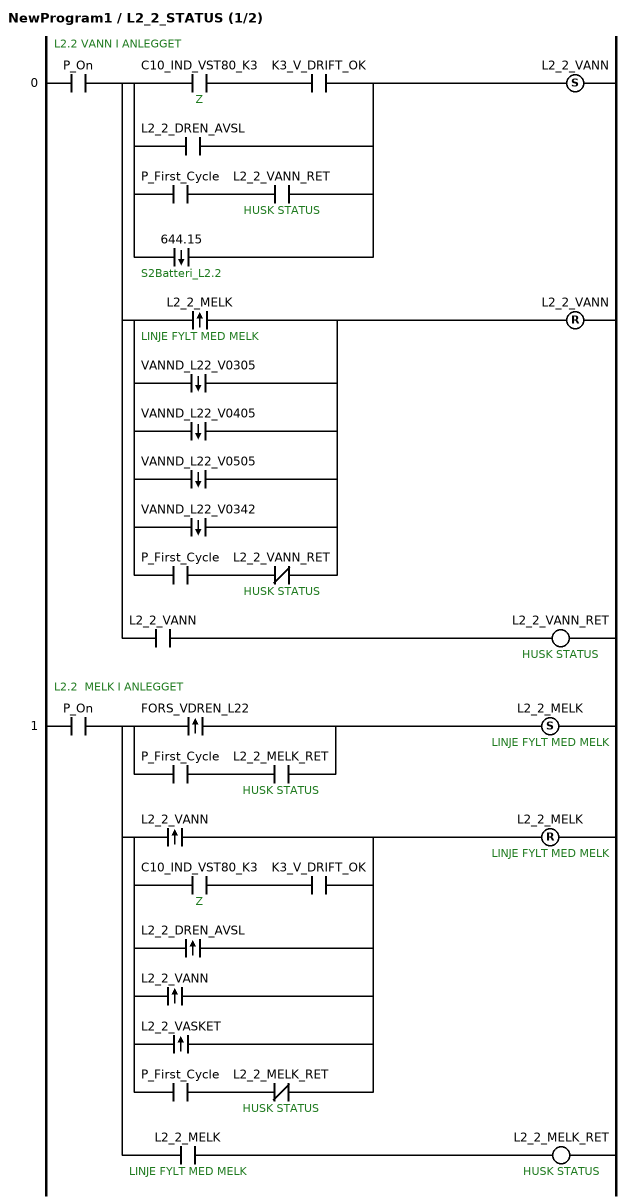
; [picture p816: NewProgram1 / L2_2_STATUS, rungs 0-1]
; rung 0: L2.2 VANN I ANLEGGET
LD P_On
OUT TR0
LD C10_IND_VST80_K3  ; Z
AND K3_V_DRIFT_OK
OR L2_2_DREN_AVSL
LD P_First_Cycle
AND L2_2_VANN_RET  ; HUSK STATUS
ORLD
%OR 644.15  ; S2Batteri_L2.2
ANDLD
SET L2_2_VANN
LD TR0
@LD L2_2_MELK  ; LINJE FYLT MED MELK
%OR VANND_L22_V0305
%OR VANND_L22_V0405
%OR VANND_L22_V0505
%OR VANND_L22_V0342
LD P_First_Cycle
ANDNOT L2_2_VANN_RET  ; HUSK STATUS
ORLD
ANDLD
RSET L2_2_VANN
LD TR0
AND L2_2_VANN
OUT L2_2_VANN_RET  ; HUSK STATUS
; rung 1: L2.2  MELK I ANLEGGET
LD P_On
OUT TR0
@LD FORS_VDREN_L22
LD P_First_Cycle
AND L2_2_MELK_RET  ; HUSK STATUS
ORLD
ANDLD
SET L2_2_MELK  ; LINJE FYLT MED MELK
LD TR0
@LD L2_2_VANN
LD C10_IND_VST80_K3  ; Z
AND K3_V_DRIFT_OK
ORLD
@OR L2_2_DREN_AVSL
@OR L2_2_VANN
@OR L2_2_VASKET
LD P_First_Cycle
ANDNOT L2_2_MELK_RET  ; HUSK STATUS
ORLD
ANDLD
RSET L2_2_MELK  ; LINJE FYLT MED MELK
LD TR0
AND L2_2_MELK  ; LINJE FYLT MED MELK
OUT L2_2_MELK_RET  ; HUSK STATUS

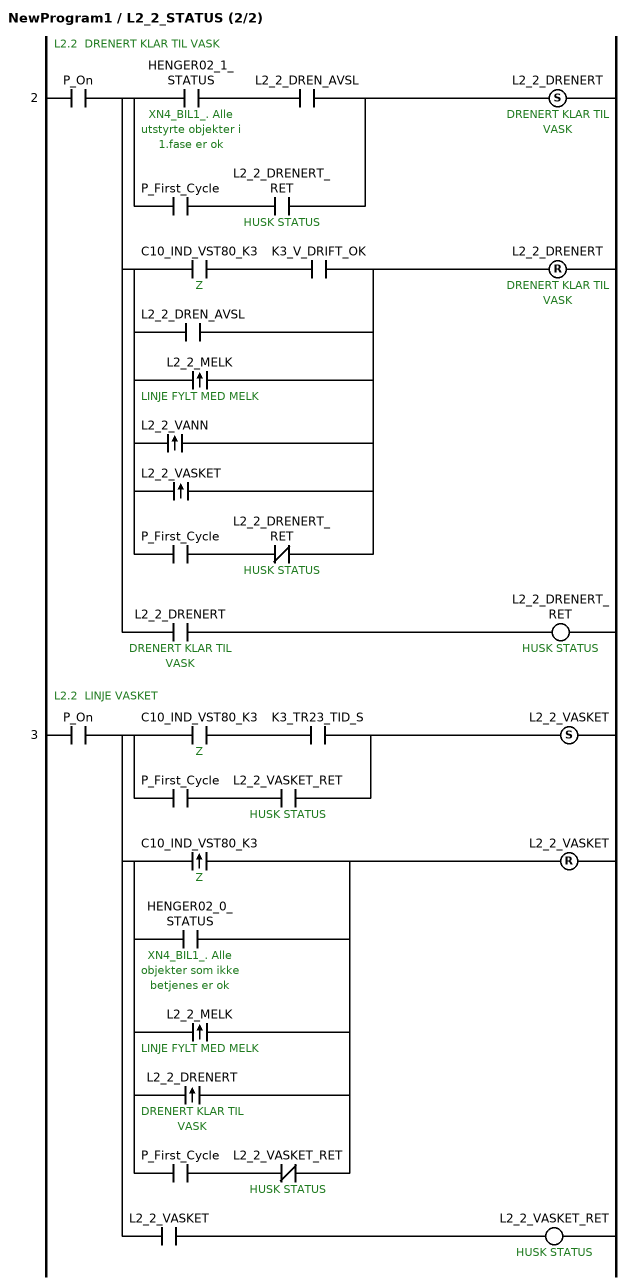
; rung 2: L2.2  DRENERT KLAR TIL VASK
LD P_On
OUT TR0
LD HENGER02_1_STATUS  ; XN4_BIL1_. Alle utstyrte objekter i 1.fase er ok
AND L2_2_DREN_AVSL
LD P_First_Cycle
AND L2_2_DRENERT_RET  ; HUSK STATUS
ORLD
ANDLD
SET L2_2_DRENERT  ; DRENERT KLAR TIL VASK
LD TR0
LD C10_IND_VST80_K3  ; Z
AND K3_V_DRIFT_OK
OR L2_2_DREN_AVSL
@OR L2_2_MELK  ; LINJE FYLT MED MELK
@OR L2_2_VANN
@OR L2_2_VASKET
LD P_First_Cycle
ANDNOT L2_2_DRENERT_RET  ; HUSK STATUS
ORLD
ANDLD
RSET L2_2_DRENERT  ; DRENERT KLAR TIL VASK
LD TR0
AND L2_2_DRENERT  ; DRENERT KLAR TIL VASK
OUT L2_2_DRENERT_RET  ; HUSK STATUS
; rung 3: L2.2  LINJE VASKET
LD P_On
OUT TR0
LD C10_IND_VST80_K3  ; Z
AND K3_TR23_TID_S
LD P_First_Cycle
AND L2_2_VASKET_RET  ; HUSK STATUS
ORLD
ANDLD
SET L2_2_VASKET
LD TR0
@LD C10_IND_VST80_K3  ; Z
OR HENGER02_0_STATUS  ; XN4_BIL1_. Alle objekter som ikke betjenes er ok
@OR L2_2_MELK  ; LINJE FYLT MED MELK
@OR L2_2_DRENERT  ; DRENERT KLAR TIL VASK
LD P_First_Cycle
ANDNOT L2_2_VASKET_RET  ; HUSK STATUS
ORLD
ANDLD
RSET L2_2_VASKET
LD TR0
AND L2_2_VASKET
OUT L2_2_VASKET_RET  ; HUSK STATUS

### Section L2_2_FUNKSJONER

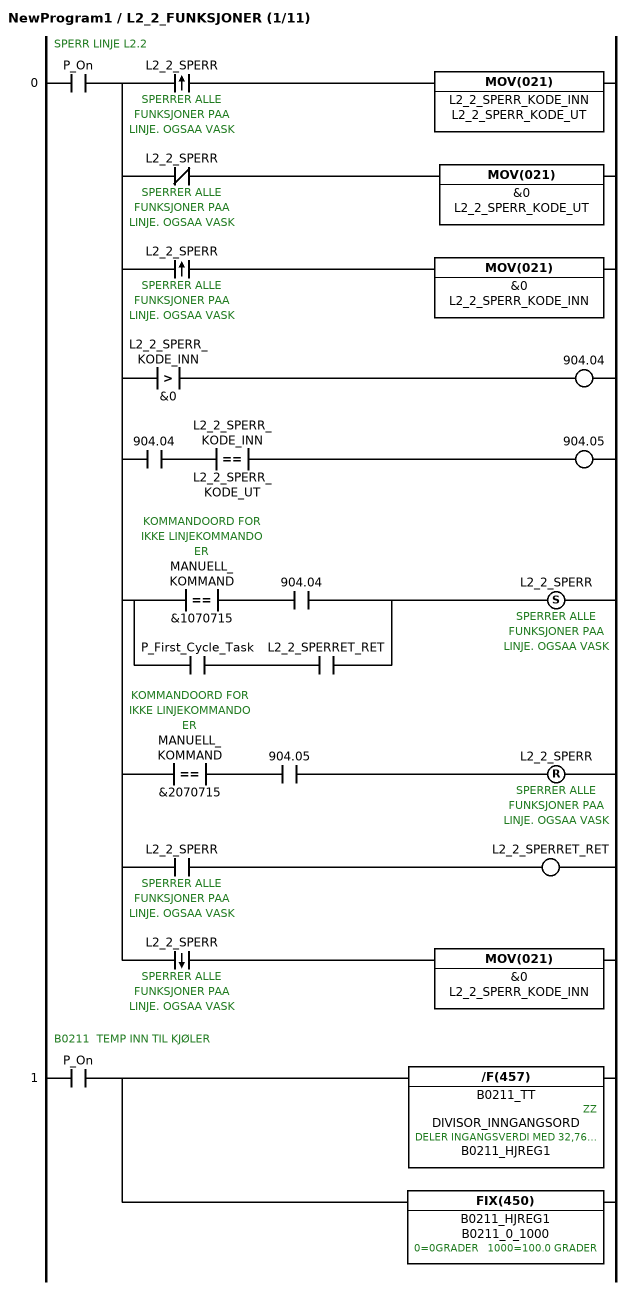
; rung 0: SPERR LINJE L2.2
LD P_On
OUT TR0
@AND L2_2_SPERR  ; SPERRER ALLE FUNKSJONER PAA LINJE. OGSAA VASK
MOV(021) L2_2_SPERR_KODE_INN L2_2_SPERR_KODE_UT
LD TR0
ANDNOT L2_2_SPERR  ; SPERRER ALLE FUNKSJONER PAA LINJE. OGSAA VASK
MOV(021) &0 L2_2_SPERR_KODE_UT
LD TR0
@AND L2_2_SPERR  ; SPERRER ALLE FUNKSJONER PAA LINJE. OGSAA VASK
MOV(021) &0 L2_2_SPERR_KODE_INN
LD TR0
AND>(320) L2_2_SPERR_KODE_INN &0
OUT 904.04
LD TR0
AND 904.04
AND=(300) L2_2_SPERR_KODE_INN L2_2_SPERR_KODE_UT
OUT 904.05
LD TR0
LD=L(301) MANUELL_KOMMAND &1070715  ; KOMMANDOORD FOR IKKE LINJEKOMMANDOER
AND 904.04
LD P_First_Cycle_Task
AND L2_2_SPERRET_RET
ORLD
ANDLD
SET L2_2_SPERR  ; SPERRER ALLE FUNKSJONER PAA LINJE. OGSAA VASK
LD TR0
AND=L(301) MANUELL_KOMMAND &2070715  ; KOMMANDOORD FOR IKKE LINJEKOMMANDOER
AND 904.05
RSET L2_2_SPERR  ; SPERRER ALLE FUNKSJONER PAA LINJE. OGSAA VASK
LD TR0
AND L2_2_SPERR  ; SPERRER ALLE FUNKSJONER PAA LINJE. OGSAA VASK
OUT L2_2_SPERRET_RET
LD TR0
%AND L2_2_SPERR  ; SPERRER ALLE FUNKSJONER PAA LINJE. OGSAA VASK
MOV(021) &0 L2_2_SPERR_KODE_INN
; rung 1: B0211  TEMP INN TIL KJØLER
LD P_On
/F(457) B0211_TT DIVISOR_INNGANGSORD B0211_HJREG1  ; ZZ, DELER INGANGSVERDI MED 32,760 FOR OMREGNING TIL 0-1000
FIX(450) B0211_HJREG1 B0211_0_1000  ; 0=0GRADER   1000=100.0 GRADER

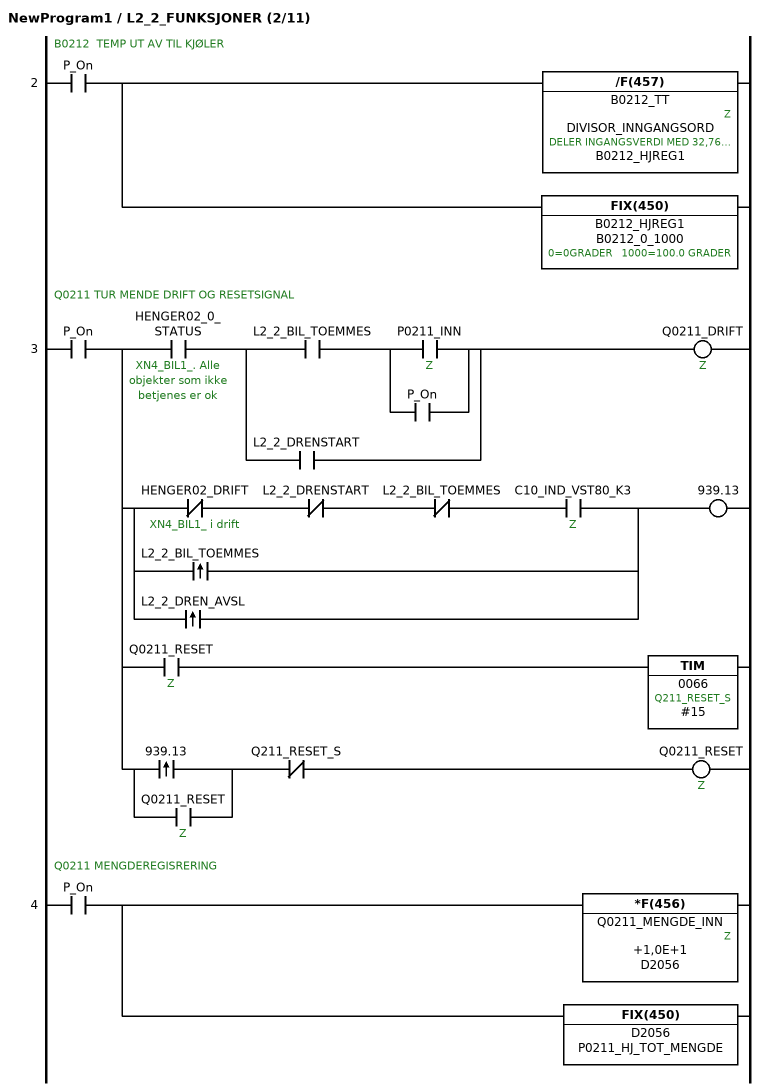
; rung 2: B0212  TEMP UT AV TIL KJØLER
LD P_On
/F(457) B0212_TT DIVISOR_INNGANGSORD B0212_HJREG1  ; Z, DELER INGANGSVERDI MED 32,760 FOR OMREGNING TIL 0-1000
FIX(450) B0212_HJREG1 B0212_0_1000  ; 0=0GRADER   1000=100.0 GRADER
; rung 3: Q0211 TUR MENDE DRIFT OG RESETSIGNAL
LD P_On
OUT TR0
AND HENGER02_0_STATUS  ; XN4_BIL1_. Alle objekter som ikke betjenes er ok
LD L2_2_BIL_TOEMMES
LD P0211_INN  ; Z
OR P_On
ANDLD
OR L2_2_DRENSTART
ANDLD
OUT Q0211_DRIFT  ; Z
LD TR0
LDNOT HENGER02_DRIFT  ; XN4_BIL1_ i drift
ANDNOT L2_2_DRENSTART
ANDNOT L2_2_BIL_TOEMMES
AND C10_IND_VST80_K3  ; Z
@OR L2_2_BIL_TOEMMES
@OR L2_2_DREN_AVSL
ANDLD
OUT 939.13
LD TR0
AND Q0211_RESET  ; Z
TIM 0066 #15  ; Q211_RESET_S
LD TR0
@LD 939.13
OR Q0211_RESET  ; Z
ANDLD
ANDNOT Q211_RESET_S
OUT Q0211_RESET  ; Z
; rung 4: Q0211 MENGDEREGISRERING
LD P_On
*F(456) Q0211_MENGDE_INN +1,0E+1 D2056  ; Z
FIX(450) D2056 P0211_HJ_TOT_MENGDE

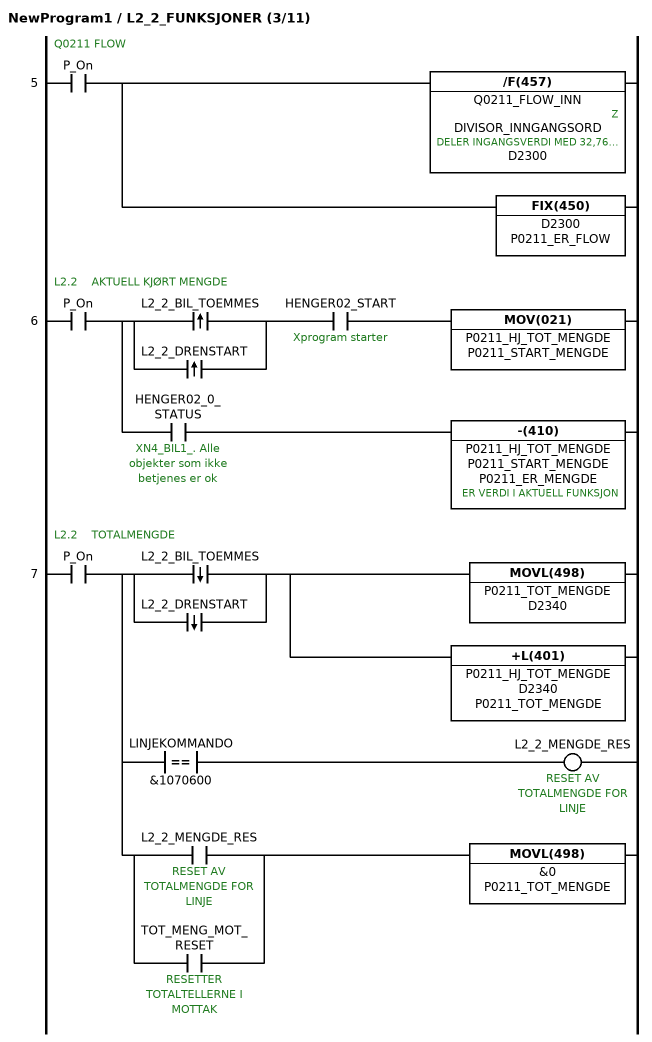
; rung 5: Q0211 FLOW
LD P_On
/F(457) Q0211_FLOW_INN DIVISOR_INNGANGSORD D2300  ; Z, DELER INGANGSVERDI MED 32,760 FOR OMREGNING TIL 0-1000
FIX(450) D2300 P0211_ER_FLOW
; rung 6: L2.2    AKTUELL KJØRT MENGDE
LD P_On
OUT TR0
@LD L2_2_BIL_TOEMMES
@OR L2_2_DRENSTART
ANDLD
AND HENGER02_START  ; Xprogram starter
MOV(021) P0211_HJ_TOT_MENGDE P0211_START_MENGDE
LD TR0
AND HENGER02_0_STATUS  ; XN4_BIL1_. Alle objekter som ikke betjenes er ok
-(410) P0211_HJ_TOT_MENGDE P0211_START_MENGDE P0211_ER_MENGDE  ; ER VERDI I AKTUELL FUNKSJON
; rung 7: L2.2    TOTALMENGDE
LD P_On
OUT TR0
%LD L2_2_BIL_TOEMMES
%OR L2_2_DRENSTART
ANDLD
MOVL(498) P0211_TOT_MENGDE D2340
+L(401) P0211_HJ_TOT_MENGDE D2340 P0211_TOT_MENGDE
LD TR0
AND=L(301) LINJEKOMMANDO &1070600
OUT L2_2_MENGDE_RES  ; RESET AV  TOTALMENGDE FOR LINJE
LD TR0
LD L2_2_MENGDE_RES  ; RESET AV  TOTALMENGDE FOR LINJE
OR TOT_MENG_MOT_RESET  ; RESETTER TOTALTELLERNE I MOTTAK
ANDLD
MOVL(498) &0 P0211_TOT_MENGDE

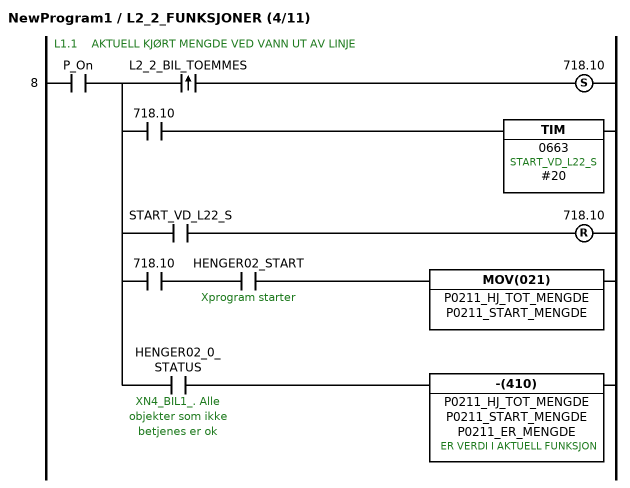
; rung 8: L1.1    AKTUELL KJØRT MENGDE VED VANN UT AV LINJE
LD P_On
OUT TR0
@AND L2_2_BIL_TOEMMES
SET 718.10
LD TR0
AND 718.10
TIM 0663 #20  ; START_VD_L22_S
LD TR0
AND START_VD_L22_S
RSET 718.10
LD TR0
AND 718.10
AND HENGER02_START  ; Xprogram starter
MOV(021) P0211_HJ_TOT_MENGDE P0211_START_MENGDE
LD TR0
AND HENGER02_0_STATUS  ; XN4_BIL1_. Alle objekter som ikke betjenes er ok
-(410) P0211_HJ_TOT_MENGDE P0211_START_MENGDE P0211_ER_MENGDE  ; ER VERDI I AKTUELL FUNKSJON

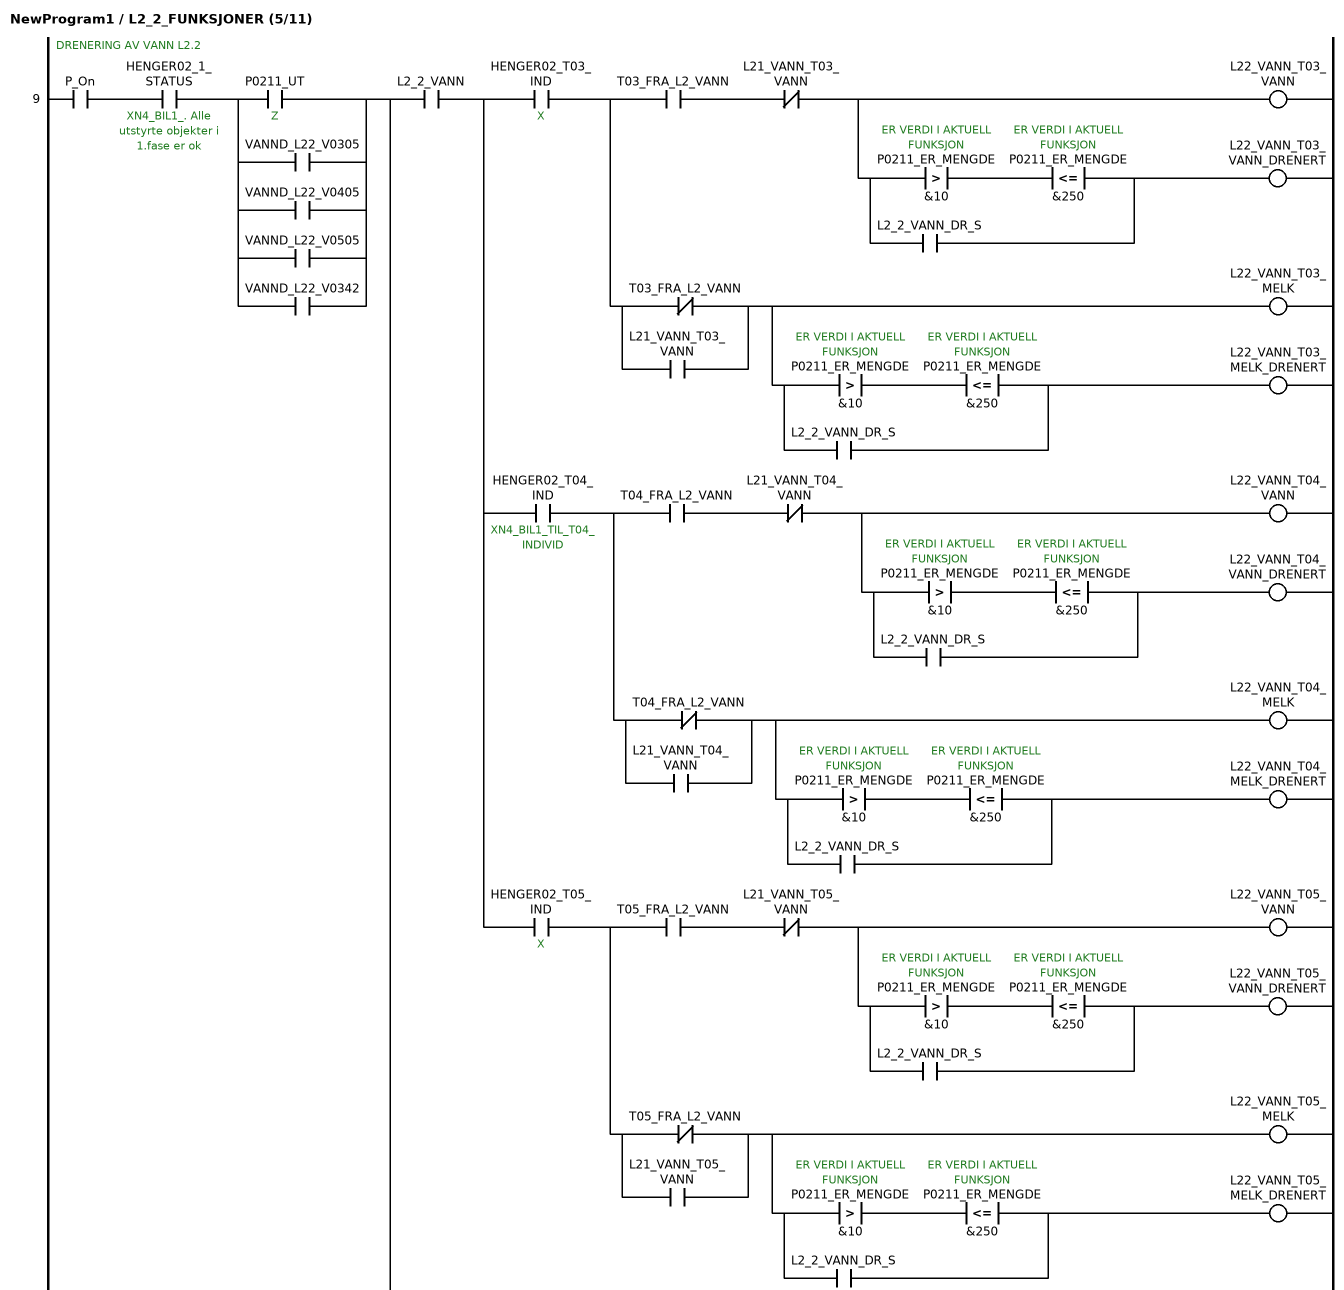

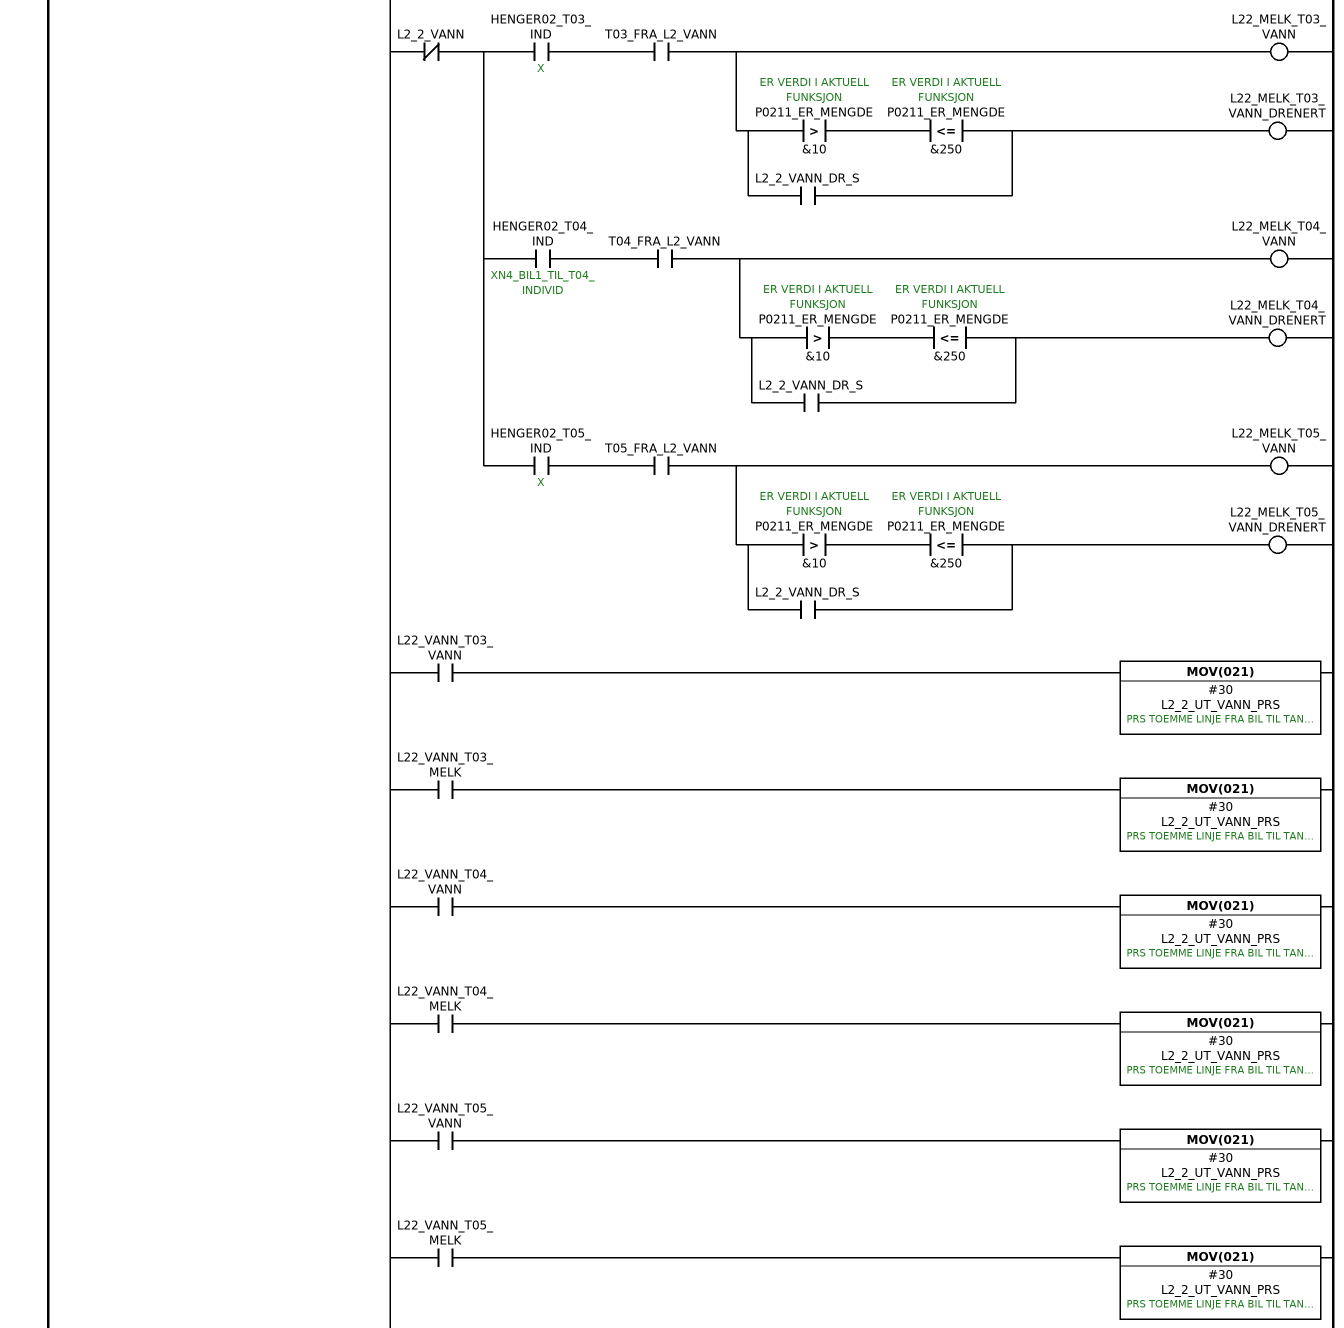

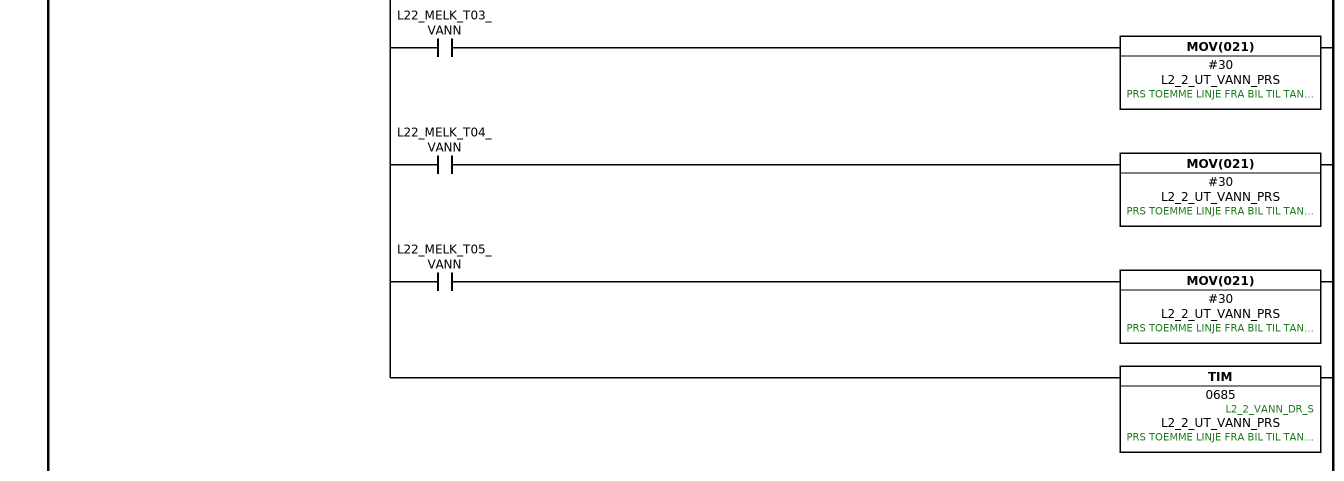
; rung 9: DRENERING AV VANN L2.2
LD P_On
AND HENGER02_1_STATUS  ; XN4_BIL1_. Alle utstyrte objekter i 1.fase er ok
LD P0211_UT  ; Z
OR VANND_L22_V0305
OR VANND_L22_V0405
OR VANND_L22_V0505
OR VANND_L22_V0342
ANDLD
OUT TR0
AND L2_2_VANN
OUT TR1
AND HENGER02_T03_IND  ; X
OUT TR2
AND T03_FRA_L2_VANN
ANDNOT L21_VANN_T03_VANN
OUT L22_VANN_T03_VANN
LD>(320) P0211_ER_MENGDE &10  ; ER VERDI I AKTUELL FUNKSJON
AND<=(315) P0211_ER_MENGDE &250  ; ER VERDI I AKTUELL FUNKSJON
OR L2_2_VANN_DR_S
ANDLD
OUT L22_VANN_T03_VANN_DRENERT
LD TR2
LDNOT T03_FRA_L2_VANN
OR L21_VANN_T03_VANN
ANDLD
OUT L22_VANN_T03_MELK
LD>(320) P0211_ER_MENGDE &10  ; ER VERDI I AKTUELL FUNKSJON
AND<=(315) P0211_ER_MENGDE &250  ; ER VERDI I AKTUELL FUNKSJON
OR L2_2_VANN_DR_S
ANDLD
OUT L22_VANN_T03_MELK_DRENERT
LD TR1
AND HENGER02_T04_IND  ; XN4_BIL1_TIL_T04_INDIVID
OUT TR2
AND T04_FRA_L2_VANN
ANDNOT L21_VANN_T04_VANN
OUT L22_VANN_T04_VANN
LD>(320) P0211_ER_MENGDE &10  ; ER VERDI I AKTUELL FUNKSJON
AND<=(315) P0211_ER_MENGDE &250  ; ER VERDI I AKTUELL FUNKSJON
OR L2_2_VANN_DR_S
ANDLD
OUT L22_VANN_T04_VANN_DRENERT
LD TR2
LDNOT T04_FRA_L2_VANN
OR L21_VANN_T04_VANN
ANDLD
OUT L22_VANN_T04_MELK
LD>(320) P0211_ER_MENGDE &10  ; ER VERDI I AKTUELL FUNKSJON
AND<=(315) P0211_ER_MENGDE &250  ; ER VERDI I AKTUELL FUNKSJON
OR L2_2_VANN_DR_S
ANDLD
OUT L22_VANN_T04_MELK_DRENERT
LD TR1
AND HENGER02_T05_IND  ; X
OUT TR1
AND T05_FRA_L2_VANN
ANDNOT L21_VANN_T05_VANN
OUT L22_VANN_T05_VANN
LD>(320) P0211_ER_MENGDE &10  ; ER VERDI I AKTUELL FUNKSJON
AND<=(315) P0211_ER_MENGDE &250  ; ER VERDI I AKTUELL FUNKSJON
OR L2_2_VANN_DR_S
ANDLD
OUT L22_VANN_T05_VANN_DRENERT
LD TR1
LDNOT T05_FRA_L2_VANN
OR L21_VANN_T05_VANN
ANDLD
OUT L22_VANN_T05_MELK
LD>(320) P0211_ER_MENGDE &10  ; ER VERDI I AKTUELL FUNKSJON
AND<=(315) P0211_ER_MENGDE &250  ; ER VERDI I AKTUELL FUNKSJON
OR L2_2_VANN_DR_S
ANDLD
OUT L22_VANN_T05_MELK_DRENERT
LD TR0
ANDNOT L2_2_VANN
OUT TR1
AND HENGER02_T03_IND  ; X
AND T03_FRA_L2_VANN
OUT L22_MELK_T03_VANN
LD>(320) P0211_ER_MENGDE &10  ; ER VERDI I AKTUELL FUNKSJON
AND<=(315) P0211_ER_MENGDE &250  ; ER VERDI I AKTUELL FUNKSJON
OR L2_2_VANN_DR_S
ANDLD
OUT L22_MELK_T03_VANN_DRENERT
LD TR1
AND HENGER02_T04_IND  ; XN4_BIL1_TIL_T04_INDIVID
AND T04_FRA_L2_VANN
OUT L22_MELK_T04_VANN
LD>(320) P0211_ER_MENGDE &10  ; ER VERDI I AKTUELL FUNKSJON
AND<=(315) P0211_ER_MENGDE &250  ; ER VERDI I AKTUELL FUNKSJON
OR L2_2_VANN_DR_S
ANDLD
OUT L22_MELK_T04_VANN_DRENERT
LD TR1
AND HENGER02_T05_IND  ; X
AND T05_FRA_L2_VANN
OUT L22_MELK_T05_VANN
LD>(320) P0211_ER_MENGDE &10  ; ER VERDI I AKTUELL FUNKSJON
AND<=(315) P0211_ER_MENGDE &250  ; ER VERDI I AKTUELL FUNKSJON
OR L2_2_VANN_DR_S
ANDLD
OUT L22_MELK_T05_VANN_DRENERT
LD TR0
AND L22_VANN_T03_VANN
MOV(021) #30 L2_2_UT_VANN_PRS  ; PRS TOEMME LINJE FRA BIL TIL TANK FOR VANN
LD TR0
AND L22_VANN_T03_MELK
MOV(021) #30 L2_2_UT_VANN_PRS  ; PRS TOEMME LINJE FRA BIL TIL TANK FOR VANN
LD TR0
AND L22_VANN_T04_VANN
MOV(021) #30 L2_2_UT_VANN_PRS  ; PRS TOEMME LINJE FRA BIL TIL TANK FOR VANN
LD TR0
AND L22_VANN_T04_MELK
MOV(021) #30 L2_2_UT_VANN_PRS  ; PRS TOEMME LINJE FRA BIL TIL TANK FOR VANN
LD TR0
AND L22_VANN_T05_VANN
MOV(021) #30 L2_2_UT_VANN_PRS  ; PRS TOEMME LINJE FRA BIL TIL TANK FOR VANN
LD TR0
AND L22_VANN_T05_MELK
MOV(021) #30 L2_2_UT_VANN_PRS  ; PRS TOEMME LINJE FRA BIL TIL TANK FOR VANN
LD TR0
AND L22_MELK_T03_VANN
MOV(021) #30 L2_2_UT_VANN_PRS  ; PRS TOEMME LINJE FRA BIL TIL TANK FOR VANN
LD TR0
AND L22_MELK_T04_VANN
MOV(021) #30 L2_2_UT_VANN_PRS  ; PRS TOEMME LINJE FRA BIL TIL TANK FOR VANN
LD TR0
AND L22_MELK_T05_VANN
MOV(021) #30 L2_2_UT_VANN_PRS  ; PRS TOEMME LINJE FRA BIL TIL TANK FOR VANN
LD TR0
TIM 0685 L2_2_UT_VANN_PRS  ; PRS TOEMME LINJE FRA BIL TIL TANK FOR VANN, L2_2_VANN_DR_S

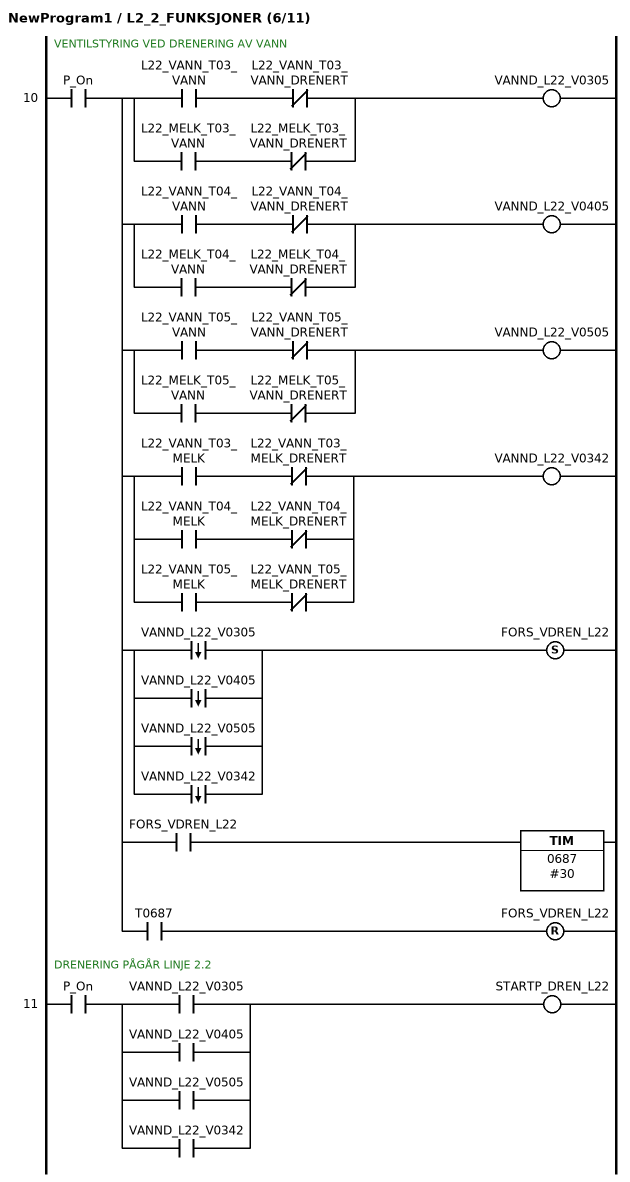
; rung 10: VENTILSTYRING VED DRENERING AV VANN
LD P_On
OUT TR0
LD L22_VANN_T03_VANN
ANDNOT L22_VANN_T03_VANN_DRENERT
LD L22_MELK_T03_VANN
ANDNOT L22_MELK_T03_VANN_DRENERT
ORLD
ANDLD
OUT VANND_L22_V0305
LD TR0
LD L22_VANN_T04_VANN
ANDNOT L22_VANN_T04_VANN_DRENERT
LD L22_MELK_T04_VANN
ANDNOT L22_MELK_T04_VANN_DRENERT
ORLD
ANDLD
OUT VANND_L22_V0405
LD TR0
LD L22_VANN_T05_VANN
ANDNOT L22_VANN_T05_VANN_DRENERT
LD L22_MELK_T05_VANN
ANDNOT L22_MELK_T05_VANN_DRENERT
ORLD
ANDLD
OUT VANND_L22_V0505
LD TR0
LD L22_VANN_T03_MELK
ANDNOT L22_VANN_T03_MELK_DRENERT
LD L22_VANN_T04_MELK
ANDNOT L22_VANN_T04_MELK_DRENERT
ORLD
LD L22_VANN_T05_MELK
ANDNOT L22_VANN_T05_MELK_DRENERT
ORLD
ANDLD
OUT VANND_L22_V0342
LD TR0
%LD VANND_L22_V0305
%OR VANND_L22_V0405
%OR VANND_L22_V0505
%OR VANND_L22_V0342
ANDLD
SET FORS_VDREN_L22
LD TR0
AND FORS_VDREN_L22
TIM 0687 #30
LD TR0
AND T0687
RSET FORS_VDREN_L22
; rung 11: DRENERING PÅGÅR LINJE 2.2
LD P_On
LD VANND_L22_V0305
OR VANND_L22_V0405
OR VANND_L22_V0505
OR VANND_L22_V0342
ANDLD
OUT STARTP_DREN_L22

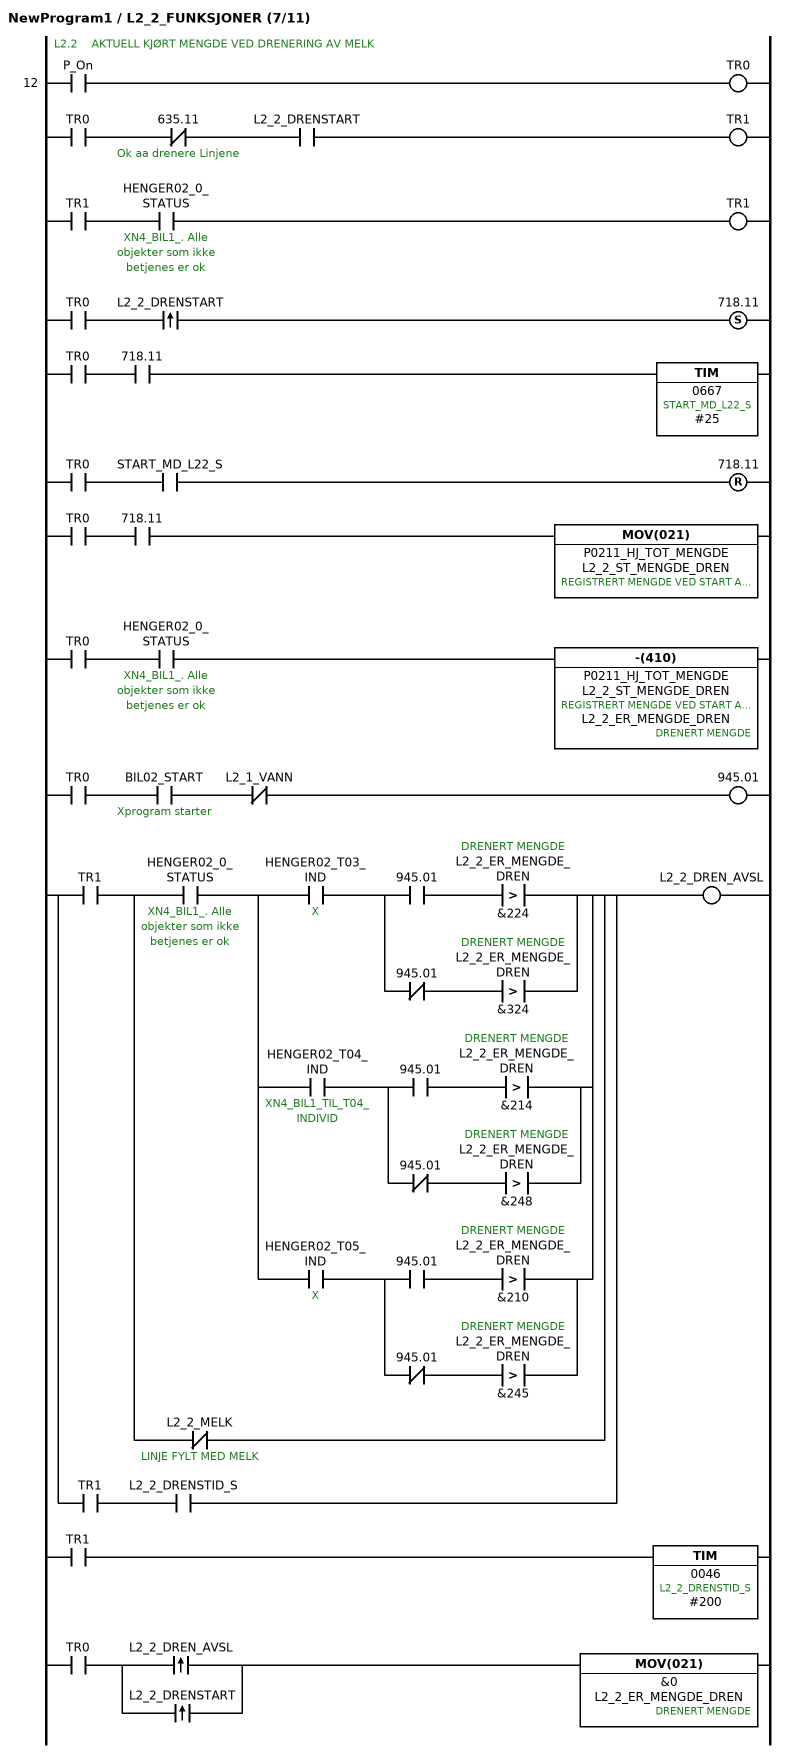
; rung 12: L2.2    AKTUELL KJØRT MENGDE VED DRENERING AV MELK
LD P_On
OUT TR0
@AND L2_2_DRENSTART
SET 718.11
LD TR0
AND 718.11
TIM 0667 #25  ; START_MD_L22_S
LD TR0
AND START_MD_L22_S
RSET 718.11
LD TR0
AND 718.11
MOV(021) P0211_HJ_TOT_MENGDE L2_2_ST_MENGDE_DREN  ; REGISTRERT MENGDE VED START AV DREN.
LD TR0
AND HENGER02_0_STATUS  ; XN4_BIL1_. Alle objekter som ikke betjenes er ok
-(410) P0211_HJ_TOT_MENGDE L2_2_ST_MENGDE_DREN L2_2_ER_MENGDE_DREN  ; REGISTRERT MENGDE VED START AV DREN., DRENERT MENGDE
LD TR0
AND BIL02_START  ; Xprogram starter
ANDNOT L2_1_VANN
OUT 945.01
LD TR0
ANDNOT 635.11  ; Ok aa drenere Linjene
AND L2_2_DRENSTART
OUT TR1
LD HENGER02_0_STATUS  ; XN4_BIL1_. Alle objekter som ikke betjenes er ok
LD HENGER02_T03_IND  ; X
LD 945.01
AND>(320) L2_2_ER_MENGDE_DREN &224  ; DRENERT MENGDE
LDNOT 945.01
AND>(320) L2_2_ER_MENGDE_DREN &324  ; DRENERT MENGDE
ORLD
ANDLD
LD HENGER02_T04_IND  ; XN4_BIL1_TIL_T04_INDIVID
LD 945.01
AND>(320) L2_2_ER_MENGDE_DREN &214  ; DRENERT MENGDE
LDNOT 945.01
AND>(320) L2_2_ER_MENGDE_DREN &248  ; DRENERT MENGDE
ORLD
ANDLD
ORLD
LD HENGER02_T05_IND  ; X
LD 945.01
AND>(320) L2_2_ER_MENGDE_DREN &210  ; DRENERT MENGDE
LDNOT 945.01
AND>(320) L2_2_ER_MENGDE_DREN &245  ; DRENERT MENGDE
ORLD
ANDLD
ORLD
ANDLD
ORNOT L2_2_MELK  ; LINJE FYLT MED MELK
ANDLD
LD TR1
AND HENGER02_0_STATUS  ; XN4_BIL1_. Alle objekter som ikke betjenes er ok
OUT TR1
AND L2_2_DRENSTID_S
ORLD
OUT L2_2_DREN_AVSL
LD TR1
TIM 0046 #200  ; L2_2_DRENSTID_S
LD TR0
@LD L2_2_DREN_AVSL
@OR L2_2_DRENSTART
ANDLD
MOV(021) &0 L2_2_ER_MENGDE_DREN  ; DRENERT MENGDE

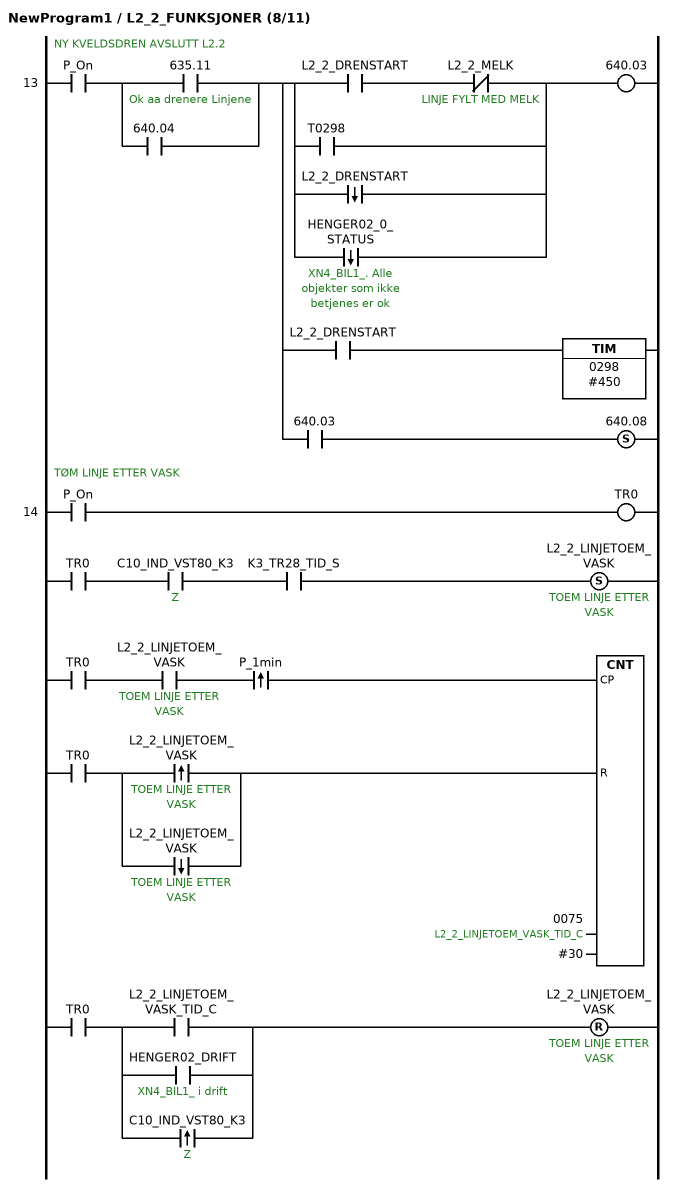
; rung 13: NY KVELDSDREN AVSLUTT L2.2
LD P_On
LD 635.11  ; Ok aa drenere Linjene
OR 640.04
ANDLD
OUT TR0
LD L2_2_DRENSTART
ANDNOT L2_2_MELK  ; LINJE FYLT MED MELK
OR T0298
%OR L2_2_DRENSTART
%OR HENGER02_0_STATUS  ; XN4_BIL1_. Alle objekter som ikke betjenes er ok
ANDLD
OUT 640.03
LD TR0
AND L2_2_DRENSTART
TIM 0298 #450
LD TR0
AND 640.03
SET 640.08
; rung 14: TØM LINJE ETTER VASK
LD P_On
OUT TR0
AND C10_IND_VST80_K3  ; Z
AND K3_TR28_TID_S
SET L2_2_LINJETOEM_VASK  ; TOEM LINJE ETTER VASK
LD TR0
AND L2_2_LINJETOEM_VASK  ; TOEM LINJE ETTER VASK
@AND P_1min
LD TR0
@LD L2_2_LINJETOEM_VASK  ; TOEM LINJE ETTER VASK
%OR L2_2_LINJETOEM_VASK  ; TOEM LINJE ETTER VASK
ANDLD
CNT 0075 #30  ; L2_2_LINJETOEM_VASK_TID_C
LD TR0
LD L2_2_LINJETOEM_VASK_TID_C
OR HENGER02_DRIFT  ; XN4_BIL1_ i drift
@OR C10_IND_VST80_K3  ; Z
ANDLD
RSET L2_2_LINJETOEM_VASK  ; TOEM LINJE ETTER VASK

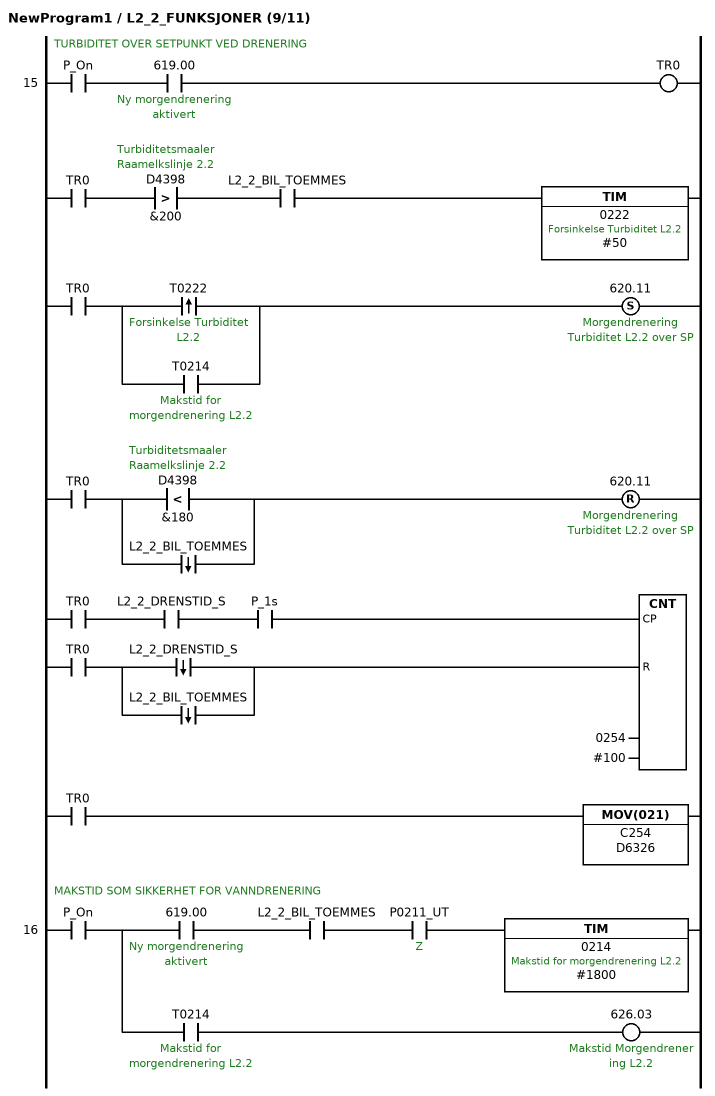
; rung 15: TURBIDITET OVER SETPUNKT VED DRENERING
LD P_On
AND 619.00  ; Ny morgendrenering aktivert
OUT TR0
AND>(320) D4398 &200  ; Turbiditetsmaaler Raamelkslinje 2.2
AND L2_2_BIL_TOEMMES
TIM 0222 #50  ; Forsinkelse Turbiditet L2.2
LD TR0
@LD T0222  ; Forsinkelse Turbiditet L2.2
OR T0214  ; Makstid for morgendrenering L2.2
ANDLD
SET 620.11  ; Morgendrenering Turbiditet L2.2 over SP
LD TR0
LD<(310) D4398 &180  ; Turbiditetsmaaler Raamelkslinje 2.2
%OR L2_2_BIL_TOEMMES
ANDLD
RSET 620.11  ; Morgendrenering Turbiditet L2.2 over SP
LD TR0
AND L2_2_DRENSTID_S
AND P_1s
LD TR0
%LD L2_2_DRENSTID_S
%OR L2_2_BIL_TOEMMES
ANDLD
CNT 0254 #100
LD TR0
MOV(021) C254 D6326
; rung 16: MAKSTID SOM SIKKERHET FOR VANNDRENERING
LD P_On
OUT TR0
AND 619.00  ; Ny morgendrenering aktivert
AND L2_2_BIL_TOEMMES
AND P0211_UT  ; Z
TIM 0214 #1800  ; Makstid for morgendrenering L2.2
LD TR0
AND T0214  ; Makstid for morgendrenering L2.2
OUT 626.03  ; Makstid Morgendrenering L2.2

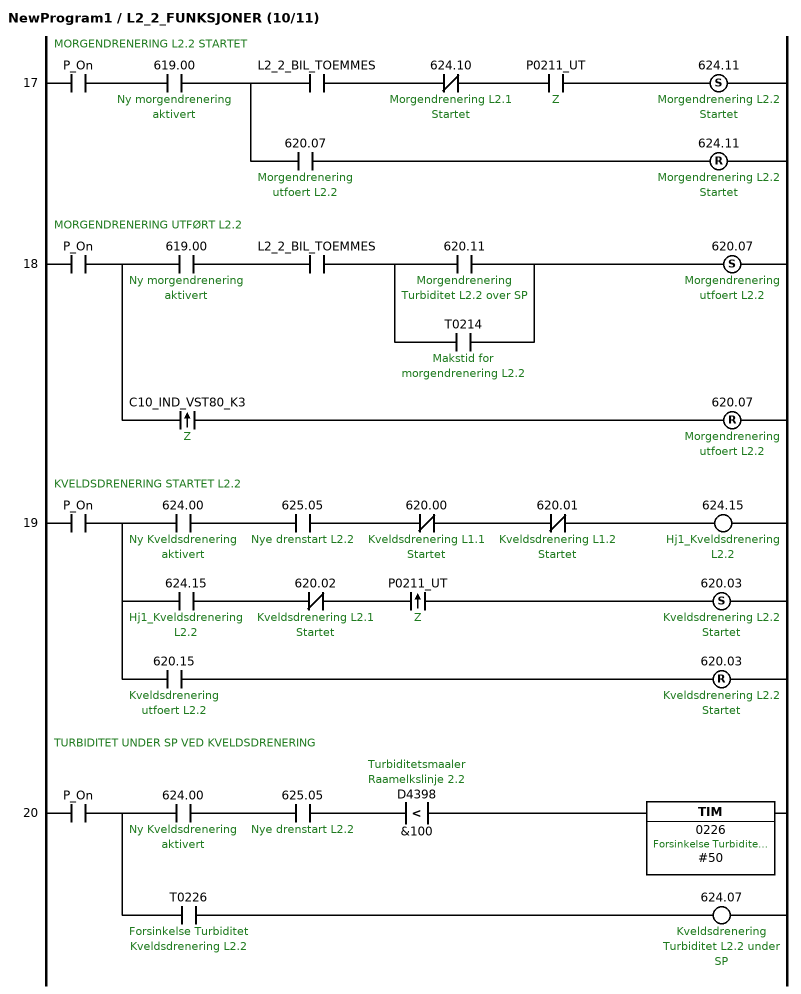
; rung 17: MORGENDRENERING L2.2 STARTET
LD P_On
AND 619.00  ; Ny morgendrenering aktivert
OUT TR0
AND L2_2_BIL_TOEMMES
ANDNOT 624.10  ; Morgendrenering L2.1 Startet
AND P0211_UT  ; Z
SET 624.11  ; Morgendrenering L2.2 Startet
LD TR0
AND 620.07  ; Morgendrenering utfoert L2.2
RSET 624.11  ; Morgendrenering L2.2 Startet
; rung 18: MORGENDRENERING UTFØRT L2.2
LD P_On
OUT TR0
AND 619.00  ; Ny morgendrenering aktivert
AND L2_2_BIL_TOEMMES
LD 620.11  ; Morgendrenering Turbiditet L2.2 over SP
OR T0214  ; Makstid for morgendrenering L2.2
ANDLD
SET 620.07  ; Morgendrenering utfoert L2.2
LD TR0
@AND C10_IND_VST80_K3  ; Z
RSET 620.07  ; Morgendrenering utfoert L2.2
; rung 19: KVELDSDRENERING STARTET L2.2
LD P_On
OUT TR0
AND 624.00  ; Ny Kveldsdrenering aktivert
AND 625.05  ; Nye drenstart L2.2
ANDNOT 620.00  ; Kveldsdrenering L1.1 Startet
ANDNOT 620.01  ; Kveldsdrenering L1.2 Startet
OUT 624.15  ; Hj1_Kveldsdrenering L2.2
LD TR0
AND 624.15  ; Hj1_Kveldsdrenering L2.2
ANDNOT 620.02  ; Kveldsdrenering L2.1 Startet
@AND P0211_UT  ; Z
SET 620.03  ; Kveldsdrenering L2.2 Startet
LD TR0
AND 620.15  ; Kveldsdrenering utfoert L2.2
RSET 620.03  ; Kveldsdrenering L2.2 Startet
; rung 20: TURBIDITET UNDER SP VED KVELDSDRENERING
LD P_On
OUT TR0
AND 624.00  ; Ny Kveldsdrenering aktivert
AND 625.05  ; Nye drenstart L2.2
AND<(310) D4398 &100  ; Turbiditetsmaaler Raamelkslinje 2.2
TIM 0226 #50  ; Forsinkelse Turbiditet Kveldsdrenering L2.2
LD TR0
AND T0226  ; Forsinkelse Turbiditet Kveldsdrenering L2.2
OUT 624.07  ; Kveldsdrenering Turbiditet L2.2 under SP

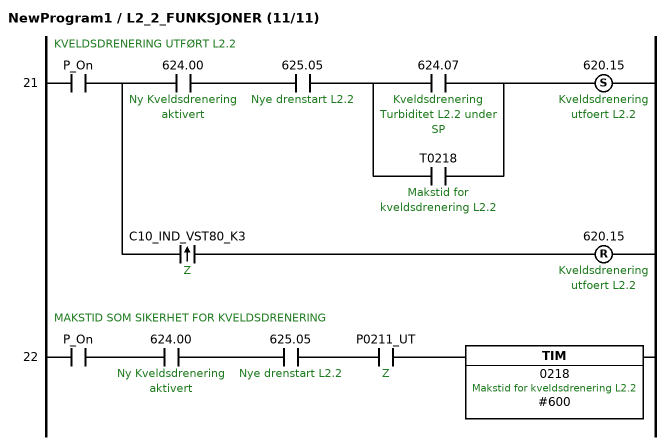
; rung 21: KVELDSDRENERING UTFØRT L2.2
LD P_On
OUT TR0
AND 624.00  ; Ny Kveldsdrenering aktivert
AND 625.05  ; Nye drenstart L2.2
LD 624.07  ; Kveldsdrenering Turbiditet L2.2 under SP
OR T0218  ; Makstid for kveldsdrenering L2.2
ANDLD
SET 620.15  ; Kveldsdrenering utfoert L2.2
LD TR0
@AND C10_IND_VST80_K3  ; Z
RSET 620.15  ; Kveldsdrenering utfoert L2.2
; rung 22: MAKSTID SOM SIKERHET FOR KVELDSDRENERING
LD P_On
AND 624.00  ; Ny Kveldsdrenering aktivert
AND 625.05  ; Nye drenstart L2.2
AND P0211_UT  ; Z
TIM 0218 #600  ; Makstid for kveldsdrenering L2.2

### Section L1_1_TIL_L2_2_FELLESFUNKSJONER

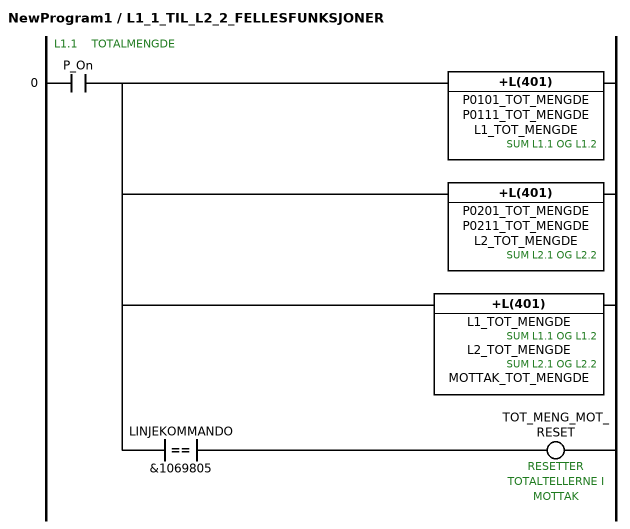
; rung 0: L1.1    TOTALMENGDE
LD P_On
+L(401) P0101_TOT_MENGDE P0111_TOT_MENGDE L1_TOT_MENGDE  ; SUM L1.1 OG L1.2
+L(401) P0201_TOT_MENGDE P0211_TOT_MENGDE L2_TOT_MENGDE  ; SUM L2.1 OG L2.2
+L(401) L1_TOT_MENGDE L2_TOT_MENGDE MOTTAK_TOT_MENGDE  ; SUM L1.1 OG L1.2, SUM L2.1 OG L2.2
AND=L(301) LINJEKOMMANDO &1069805
OUT TOT_MENG_MOT_RESET  ; RESETTER TOTALTELLERNE I MOTTAK

### Section ISVANN

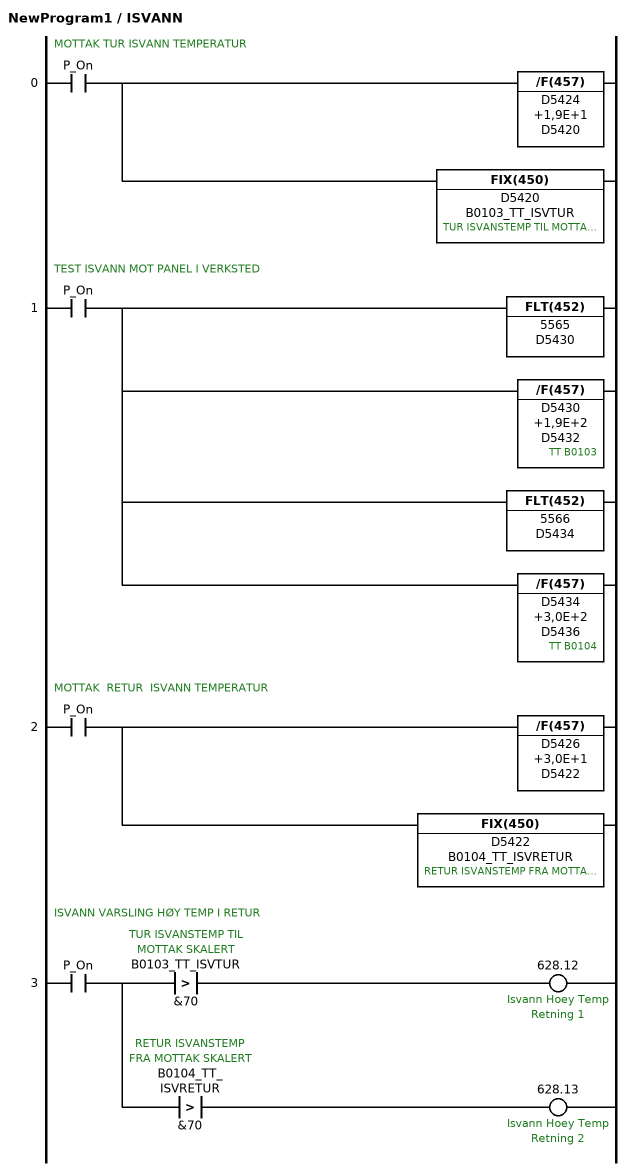
; rung 0: MOTTAK TUR ISVANN TEMPERATUR
LD P_On
/F(457) D5424 +1,9E+1 D5420
FIX(450) D5420 B0103_TT_ISVTUR  ; TUR ISVANSTEMP TIL MOTTAK SKALERT
; rung 1: TEST ISVANN MOT PANEL I VERKSTED
LD P_On
FLT(452) 5565 D5430
/F(457) D5430 +1,9E+2 D5432  ; TT B0103
FLT(452) 5566 D5434
/F(457) D5434 +3,0E+2 D5436  ; TT B0104
; rung 2: MOTTAK  RETUR  ISVANN TEMPERATUR
LD P_On
/F(457) D5426 +3,0E+1 D5422
FIX(450) D5422 B0104_TT_ISVRETUR  ; RETUR ISVANSTEMP FRA MOTTAK SKALERT
; rung 3: ISVANN VARSLING HØY TEMP I RETUR
LD P_On
OUT TR0
AND>(320) B0103_TT_ISVTUR &70  ; TUR ISVANSTEMP TIL MOTTAK SKALERT
OUT 628.12  ; Isvann Hoey Temp Retning 1
LD TR0
AND>(320) B0104_TT_ISVRETUR &70  ; RETUR ISVANSTEMP FRA MOTTAK SKALERT
OUT 628.13  ; Isvann Hoey Temp Retning 2

### Section TRYKKOVERVÅKING_RÅMELK_ISVANN

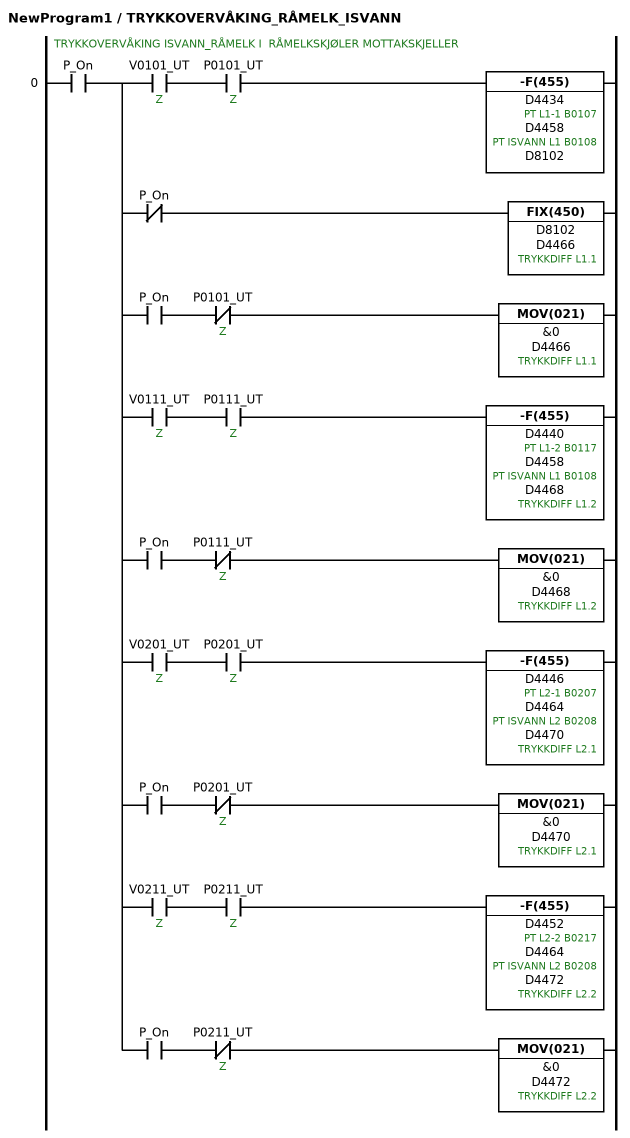
; rung 0: TRYKKOVERVÅKING ISVANN_RÅMELK I  RÅMELKSKJØLER MOTTAKSKJELLER
LD P_On
OUT TR0
AND V0101_UT  ; Z
AND P0101_UT  ; Z
-F(455) D4434 D4458 D8102  ; PT L1-1 B0107, PT ISVANN L1 B0108
LD TR0
ANDNOT P_On
FIX(450) D8102 D4466  ; TRYKKDIFF L1.1
LD TR0
AND P_On
ANDNOT P0101_UT  ; Z
MOV(021) &0 D4466  ; TRYKKDIFF L1.1
LD TR0
AND V0111_UT  ; Z
AND P0111_UT  ; Z
-F(455) D4440 D4458 D4468  ; PT L1-2 B0117, PT ISVANN L1 B0108, TRYKKDIFF L1.2
LD TR0
AND P_On
ANDNOT P0111_UT  ; Z
MOV(021) &0 D4468  ; TRYKKDIFF L1.2
LD TR0
AND V0201_UT  ; Z
AND P0201_UT  ; Z
-F(455) D4446 D4464 D4470  ; PT L2-1 B0207, PT ISVANN L2 B0208, TRYKKDIFF L2.1
LD TR0
AND P_On
ANDNOT P0201_UT  ; Z
MOV(021) &0 D4470  ; TRYKKDIFF L2.1
LD TR0
AND V0211_UT  ; Z
AND P0211_UT  ; Z
-F(455) D4452 D4464 D4472  ; PT L2-2 B0217, PT ISVANN L2 B0208, TRYKKDIFF L2.2
LD TR0
AND P_On
ANDNOT P0211_UT  ; Z
MOV(021) &0 D4472  ; TRYKKDIFF L2.2

### Section RETURPUMPER_VASKER

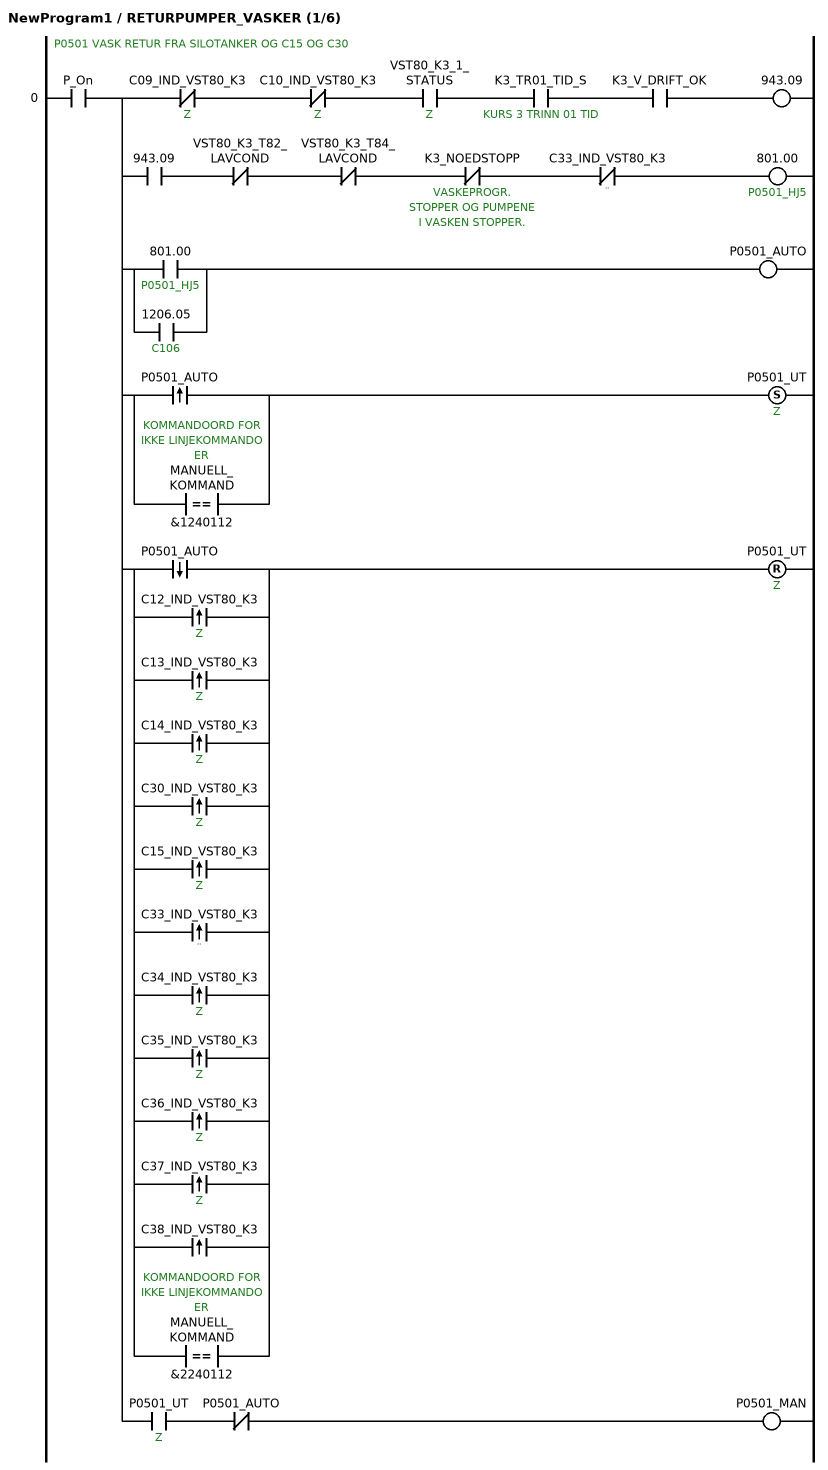
; rung 0: P0501 VASK RETUR FRA SILOTANKER OG C15 OG C30
LD P_On
OUT TR0
ANDNOT C09_IND_VST80_K3  ; Z
ANDNOT C10_IND_VST80_K3  ; Z
AND VST80_K3_1_STATUS  ; Z
AND K3_TR01_TID_S  ; KURS 3 TRINN 01 TID
AND K3_V_DRIFT_OK
OUT 943.09
LD TR0
AND 943.09
ANDNOT VST80_K3_T82_LAVCOND
ANDNOT VST80_K3_T84_LAVCOND
ANDNOT K3_NOEDSTOPP  ; VASKEPROGR. STOPPER OG PUMPENE I VASKEN STOPPER.
ANDNOT C33_IND_VST80_K3  ; ¨
OUT 801.00  ; P0501_HJ5
LD TR0
LD 801.00  ; P0501_HJ5
OR 1206.05  ; C106
ANDLD
OUT P0501_AUTO
LD TR0
@LD P0501_AUTO
OR=L(301) MANUELL_KOMMAND &1240112  ; KOMMANDOORD FOR IKKE LINJEKOMMANDOER
ANDLD
SET P0501_UT  ; Z
LD TR0
%LD P0501_AUTO
@OR C12_IND_VST80_K3  ; Z
@OR C13_IND_VST80_K3  ; Z
@OR C14_IND_VST80_K3  ; Z
@OR C30_IND_VST80_K3  ; Z
@OR C15_IND_VST80_K3  ; Z
@OR C33_IND_VST80_K3  ; ¨
@OR C34_IND_VST80_K3  ; Z
@OR C35_IND_VST80_K3  ; Z
@OR C36_IND_VST80_K3  ; Z
@OR C37_IND_VST80_K3  ; Z
@OR C38_IND_VST80_K3
OR=L(301) MANUELL_KOMMAND &2240112  ; KOMMANDOORD FOR IKKE LINJEKOMMANDOER
ANDLD
RSET P0501_UT  ; Z
LD TR0
AND P0501_UT  ; Z
ANDNOT P0501_AUTO
OUT P0501_MAN

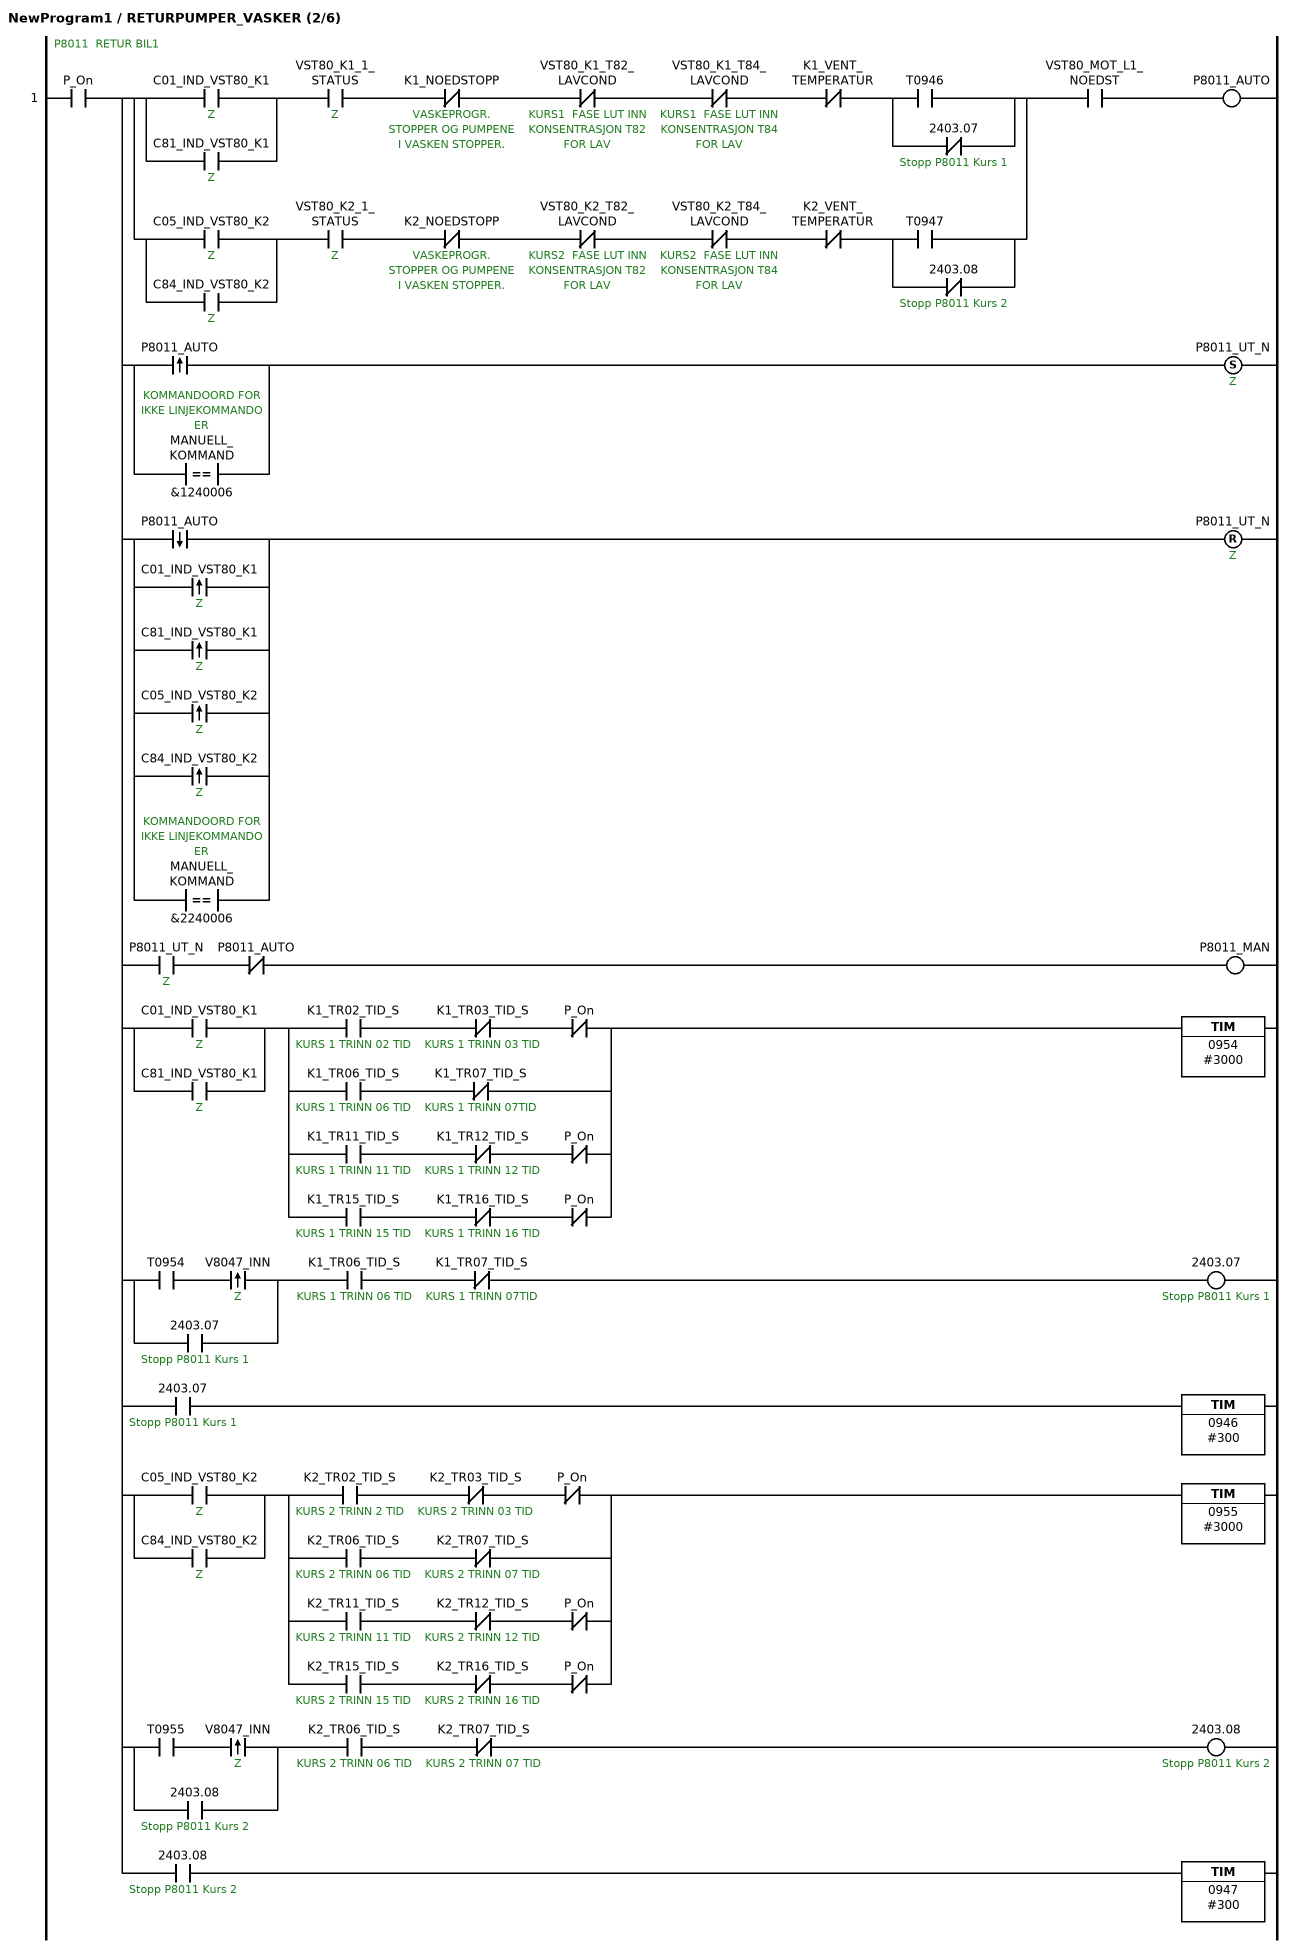
; rung 1: P8011  RETUR BIL1
LD P_On
OUT TR0
LD C01_IND_VST80_K1  ; Z
OR C81_IND_VST80_K1  ; Z
AND VST80_K1_1_STATUS  ; Z
ANDNOT K1_NOEDSTOPP  ; VASKEPROGR. STOPPER OG PUMPENE I VASKEN STOPPER.
ANDNOT VST80_K1_T82_LAVCOND  ; KURS1  FASE LUT INN KONSENTRASJON T82 FOR LAV
ANDNOT VST80_K1_T84_LAVCOND  ; KURS1  FASE LUT INN KONSENTRASJON T84 FOR LAV
ANDNOT K1_VENT_TEMPERATUR
LD T0946
ORNOT 2403.07  ; Stopp P8011 Kurs 1
ANDLD
LD C05_IND_VST80_K2  ; Z
OR C84_IND_VST80_K2  ; Z
AND VST80_K2_1_STATUS  ; Z
ANDNOT K2_NOEDSTOPP  ; VASKEPROGR. STOPPER OG PUMPENE I VASKEN STOPPER.
ANDNOT VST80_K2_T82_LAVCOND  ; KURS2  FASE LUT INN KONSENTRASJON T82 FOR LAV
ANDNOT VST80_K2_T84_LAVCOND  ; KURS2  FASE LUT INN KONSENTRASJON T84 FOR LAV
ANDNOT K2_VENT_TEMPERATUR
LD T0947
ORNOT 2403.08  ; Stopp P8011 Kurs 2
ANDLD
ORLD
ANDLD
AND VST80_MOT_L1_NOEDST
OUT P8011_AUTO
LD TR0
@LD P8011_AUTO
OR=L(301) MANUELL_KOMMAND &1240006  ; KOMMANDOORD FOR IKKE LINJEKOMMANDOER
ANDLD
SET P8011_UT_N  ; Z
LD TR0
%LD P8011_AUTO
@OR C01_IND_VST80_K1  ; Z
@OR C81_IND_VST80_K1  ; Z
@OR C05_IND_VST80_K2  ; Z
@OR C84_IND_VST80_K2  ; Z
OR=L(301) MANUELL_KOMMAND &2240006  ; KOMMANDOORD FOR IKKE LINJEKOMMANDOER
ANDLD
RSET P8011_UT_N  ; Z
LD TR0
AND P8011_UT_N  ; Z
ANDNOT P8011_AUTO
OUT P8011_MAN
LD TR0
LD C01_IND_VST80_K1  ; Z
OR C81_IND_VST80_K1  ; Z
ANDLD
LD K1_TR02_TID_S  ; KURS 1 TRINN 02 TID
ANDNOT K1_TR03_TID_S  ; KURS 1 TRINN 03 TID
ANDNOT P_On
LD K1_TR06_TID_S  ; KURS 1 TRINN 06 TID
ANDNOT K1_TR07_TID_S  ; KURS 1 TRINN 07TID
ORLD
LD K1_TR11_TID_S  ; KURS 1 TRINN 11 TID
ANDNOT K1_TR12_TID_S  ; KURS 1 TRINN 12 TID
ANDNOT P_On
ORLD
LD K1_TR15_TID_S  ; KURS 1 TRINN 15 TID
ANDNOT K1_TR16_TID_S  ; KURS 1 TRINN 16 TID
ANDNOT P_On
ORLD
ANDLD
TIM 0954 #3000
LD TR0
LD T0954
@AND V8047_INN  ; Z
OR 2403.07  ; Stopp P8011 Kurs 1
ANDLD
AND K1_TR06_TID_S  ; KURS 1 TRINN 06 TID
ANDNOT K1_TR07_TID_S  ; KURS 1 TRINN 07TID
OUT 2403.07  ; Stopp P8011 Kurs 1
LD TR0
AND 2403.07  ; Stopp P8011 Kurs 1
TIM 0946 #300
LD TR0
LD C05_IND_VST80_K2  ; Z
OR C84_IND_VST80_K2  ; Z
ANDLD
LD K2_TR02_TID_S  ; KURS 2 TRINN 2 TID
ANDNOT K2_TR03_TID_S  ; KURS 2 TRINN 03 TID
ANDNOT P_On
LD K2_TR06_TID_S  ; KURS 2 TRINN 06 TID
ANDNOT K2_TR07_TID_S  ; KURS 2 TRINN 07 TID
ORLD
LD K2_TR11_TID_S  ; KURS 2 TRINN 11 TID
ANDNOT K2_TR12_TID_S  ; KURS 2 TRINN 12 TID
ANDNOT P_On
ORLD
LD K2_TR15_TID_S  ; KURS 2 TRINN 15 TID
ANDNOT K2_TR16_TID_S  ; KURS 2 TRINN 16 TID
ANDNOT P_On
ORLD
ANDLD
TIM 0955 #3000
LD TR0
LD T0955
@AND V8047_INN  ; Z
OR 2403.08  ; Stopp P8011 Kurs 2
ANDLD
AND K2_TR06_TID_S  ; KURS 2 TRINN 06 TID
ANDNOT K2_TR07_TID_S  ; KURS 2 TRINN 07 TID
OUT 2403.08  ; Stopp P8011 Kurs 2
LD TR0
AND 2403.08  ; Stopp P8011 Kurs 2
TIM 0947 #300

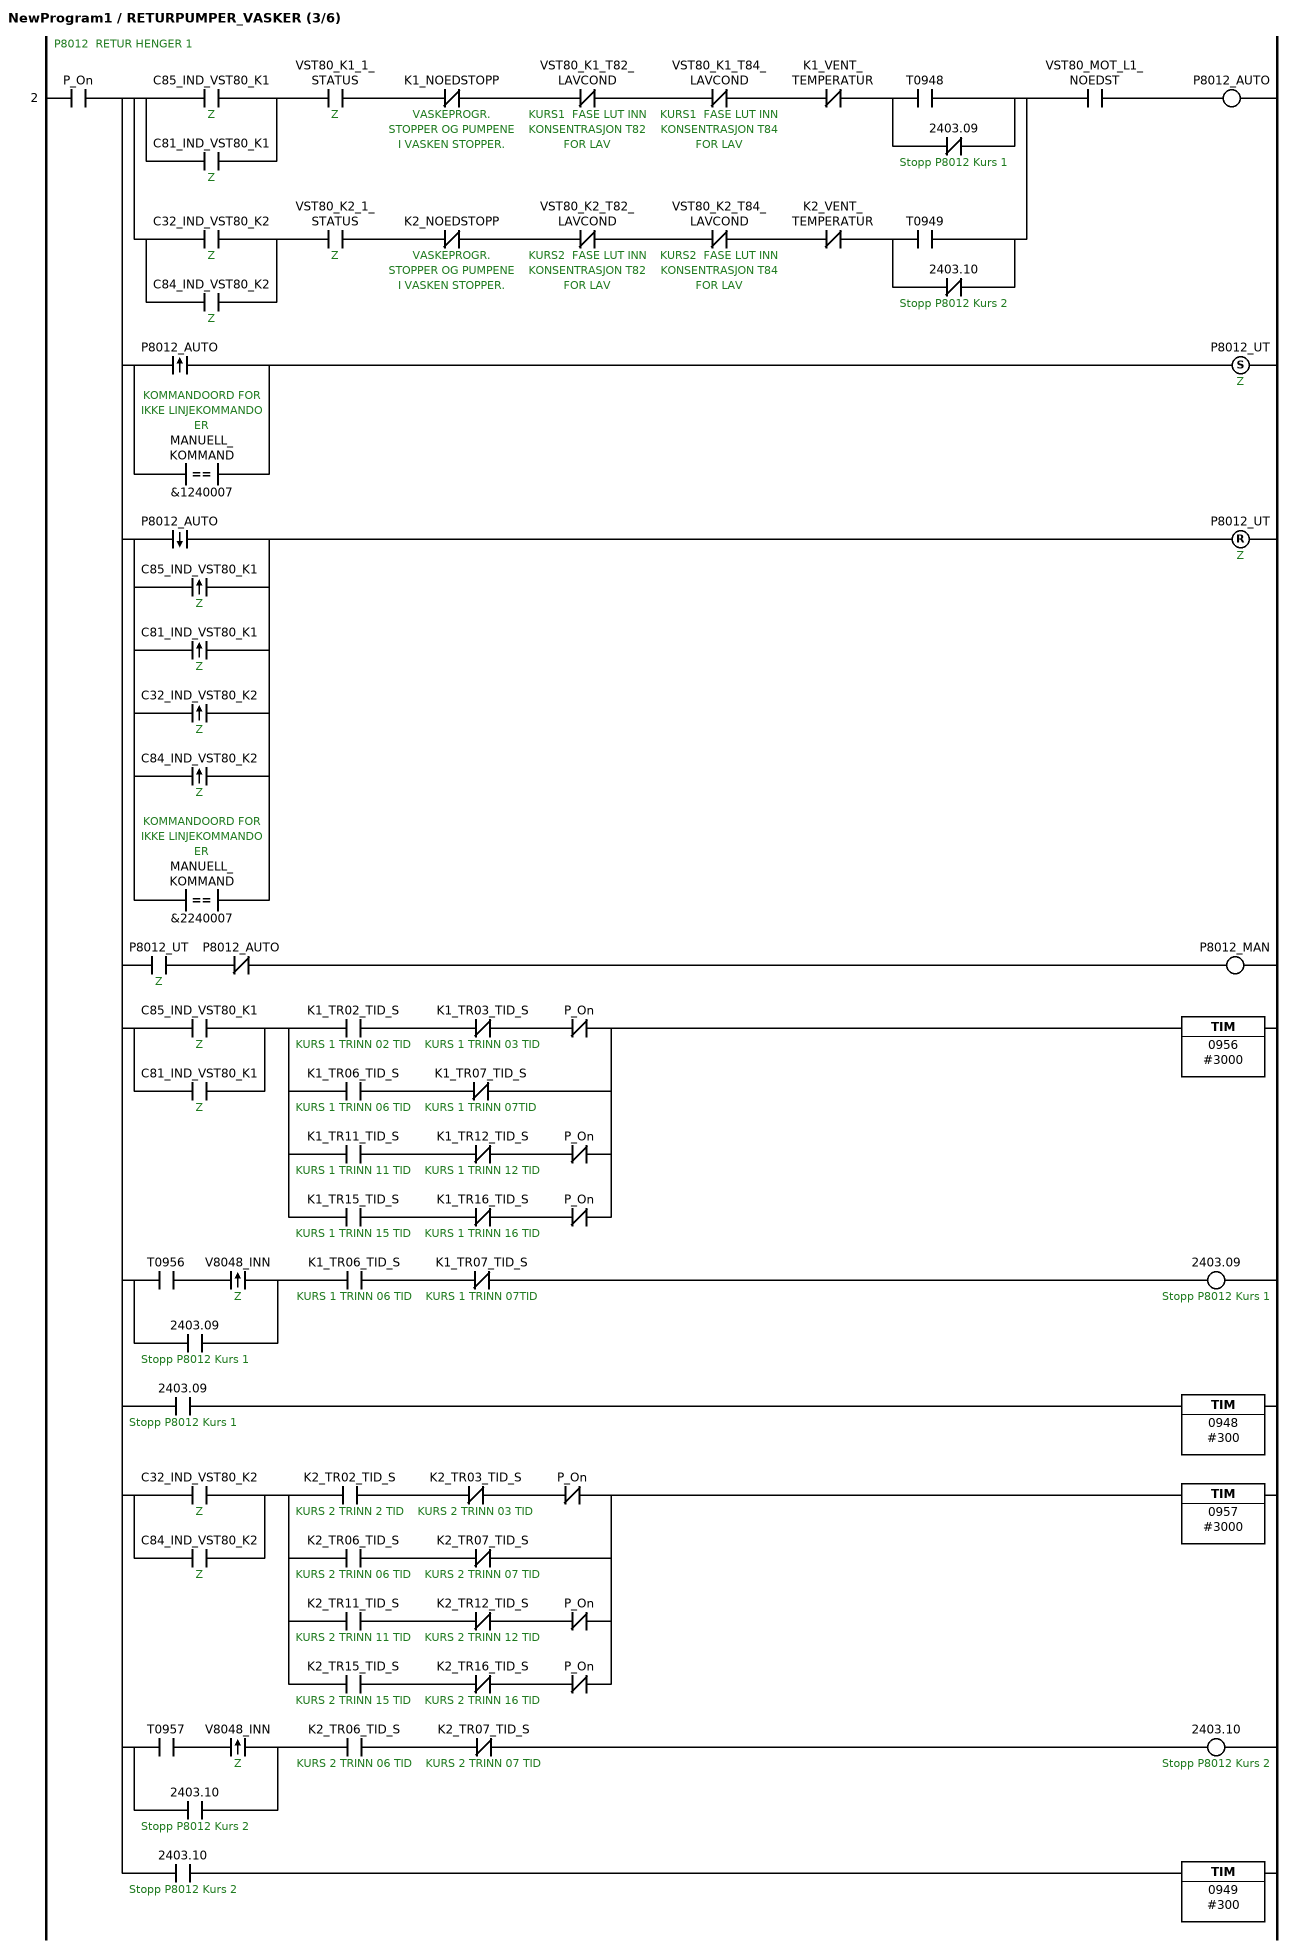
; rung 2: P8012  RETUR HENGER 1
LD P_On
OUT TR0
LD C85_IND_VST80_K1  ; Z
OR C81_IND_VST80_K1  ; Z
AND VST80_K1_1_STATUS  ; Z
ANDNOT K1_NOEDSTOPP  ; VASKEPROGR. STOPPER OG PUMPENE I VASKEN STOPPER.
ANDNOT VST80_K1_T82_LAVCOND  ; KURS1  FASE LUT INN KONSENTRASJON T82 FOR LAV
ANDNOT VST80_K1_T84_LAVCOND  ; KURS1  FASE LUT INN KONSENTRASJON T84 FOR LAV
ANDNOT K1_VENT_TEMPERATUR
LD T0948
ORNOT 2403.09  ; Stopp P8012 Kurs 1
ANDLD
LD C32_IND_VST80_K2  ; Z
OR C84_IND_VST80_K2  ; Z
AND VST80_K2_1_STATUS  ; Z
ANDNOT K2_NOEDSTOPP  ; VASKEPROGR. STOPPER OG PUMPENE I VASKEN STOPPER.
ANDNOT VST80_K2_T82_LAVCOND  ; KURS2  FASE LUT INN KONSENTRASJON T82 FOR LAV
ANDNOT VST80_K2_T84_LAVCOND  ; KURS2  FASE LUT INN KONSENTRASJON T84 FOR LAV
ANDNOT K2_VENT_TEMPERATUR
LD T0949
ORNOT 2403.10  ; Stopp P8012 Kurs 2
ANDLD
ORLD
ANDLD
AND VST80_MOT_L1_NOEDST
OUT P8012_AUTO
LD TR0
@LD P8012_AUTO
OR=L(301) MANUELL_KOMMAND &1240007  ; KOMMANDOORD FOR IKKE LINJEKOMMANDOER
ANDLD
SET P8012_UT  ; Z
LD TR0
%LD P8012_AUTO
@OR C85_IND_VST80_K1  ; Z
@OR C81_IND_VST80_K1  ; Z
@OR C32_IND_VST80_K2  ; Z
@OR C84_IND_VST80_K2  ; Z
OR=L(301) MANUELL_KOMMAND &2240007  ; KOMMANDOORD FOR IKKE LINJEKOMMANDOER
ANDLD
RSET P8012_UT  ; Z
LD TR0
AND P8012_UT  ; Z
ANDNOT P8012_AUTO
OUT P8012_MAN
LD TR0
LD C85_IND_VST80_K1  ; Z
OR C81_IND_VST80_K1  ; Z
ANDLD
LD K1_TR02_TID_S  ; KURS 1 TRINN 02 TID
ANDNOT K1_TR03_TID_S  ; KURS 1 TRINN 03 TID
ANDNOT P_On
LD K1_TR06_TID_S  ; KURS 1 TRINN 06 TID
ANDNOT K1_TR07_TID_S  ; KURS 1 TRINN 07TID
ORLD
LD K1_TR11_TID_S  ; KURS 1 TRINN 11 TID
ANDNOT K1_TR12_TID_S  ; KURS 1 TRINN 12 TID
ANDNOT P_On
ORLD
LD K1_TR15_TID_S  ; KURS 1 TRINN 15 TID
ANDNOT K1_TR16_TID_S  ; KURS 1 TRINN 16 TID
ANDNOT P_On
ORLD
ANDLD
TIM 0956 #3000
LD TR0
LD T0956
@AND V8048_INN  ; Z
OR 2403.09  ; Stopp P8012 Kurs 1
ANDLD
AND K1_TR06_TID_S  ; KURS 1 TRINN 06 TID
ANDNOT K1_TR07_TID_S  ; KURS 1 TRINN 07TID
OUT 2403.09  ; Stopp P8012 Kurs 1
LD TR0
AND 2403.09  ; Stopp P8012 Kurs 1
TIM 0948 #300
LD TR0
LD C32_IND_VST80_K2  ; Z
OR C84_IND_VST80_K2  ; Z
ANDLD
LD K2_TR02_TID_S  ; KURS 2 TRINN 2 TID
ANDNOT K2_TR03_TID_S  ; KURS 2 TRINN 03 TID
ANDNOT P_On
LD K2_TR06_TID_S  ; KURS 2 TRINN 06 TID
ANDNOT K2_TR07_TID_S  ; KURS 2 TRINN 07 TID
ORLD
LD K2_TR11_TID_S  ; KURS 2 TRINN 11 TID
ANDNOT K2_TR12_TID_S  ; KURS 2 TRINN 12 TID
ANDNOT P_On
ORLD
LD K2_TR15_TID_S  ; KURS 2 TRINN 15 TID
ANDNOT K2_TR16_TID_S  ; KURS 2 TRINN 16 TID
ANDNOT P_On
ORLD
ANDLD
TIM 0957 #3000
LD TR0
LD T0957
@AND V8048_INN  ; Z
OR 2403.10  ; Stopp P8012 Kurs 2
ANDLD
AND K2_TR06_TID_S  ; KURS 2 TRINN 06 TID
ANDNOT K2_TR07_TID_S  ; KURS 2 TRINN 07 TID
OUT 2403.10  ; Stopp P8012 Kurs 2
LD TR0
AND 2403.10  ; Stopp P8012 Kurs 2
TIM 0949 #300

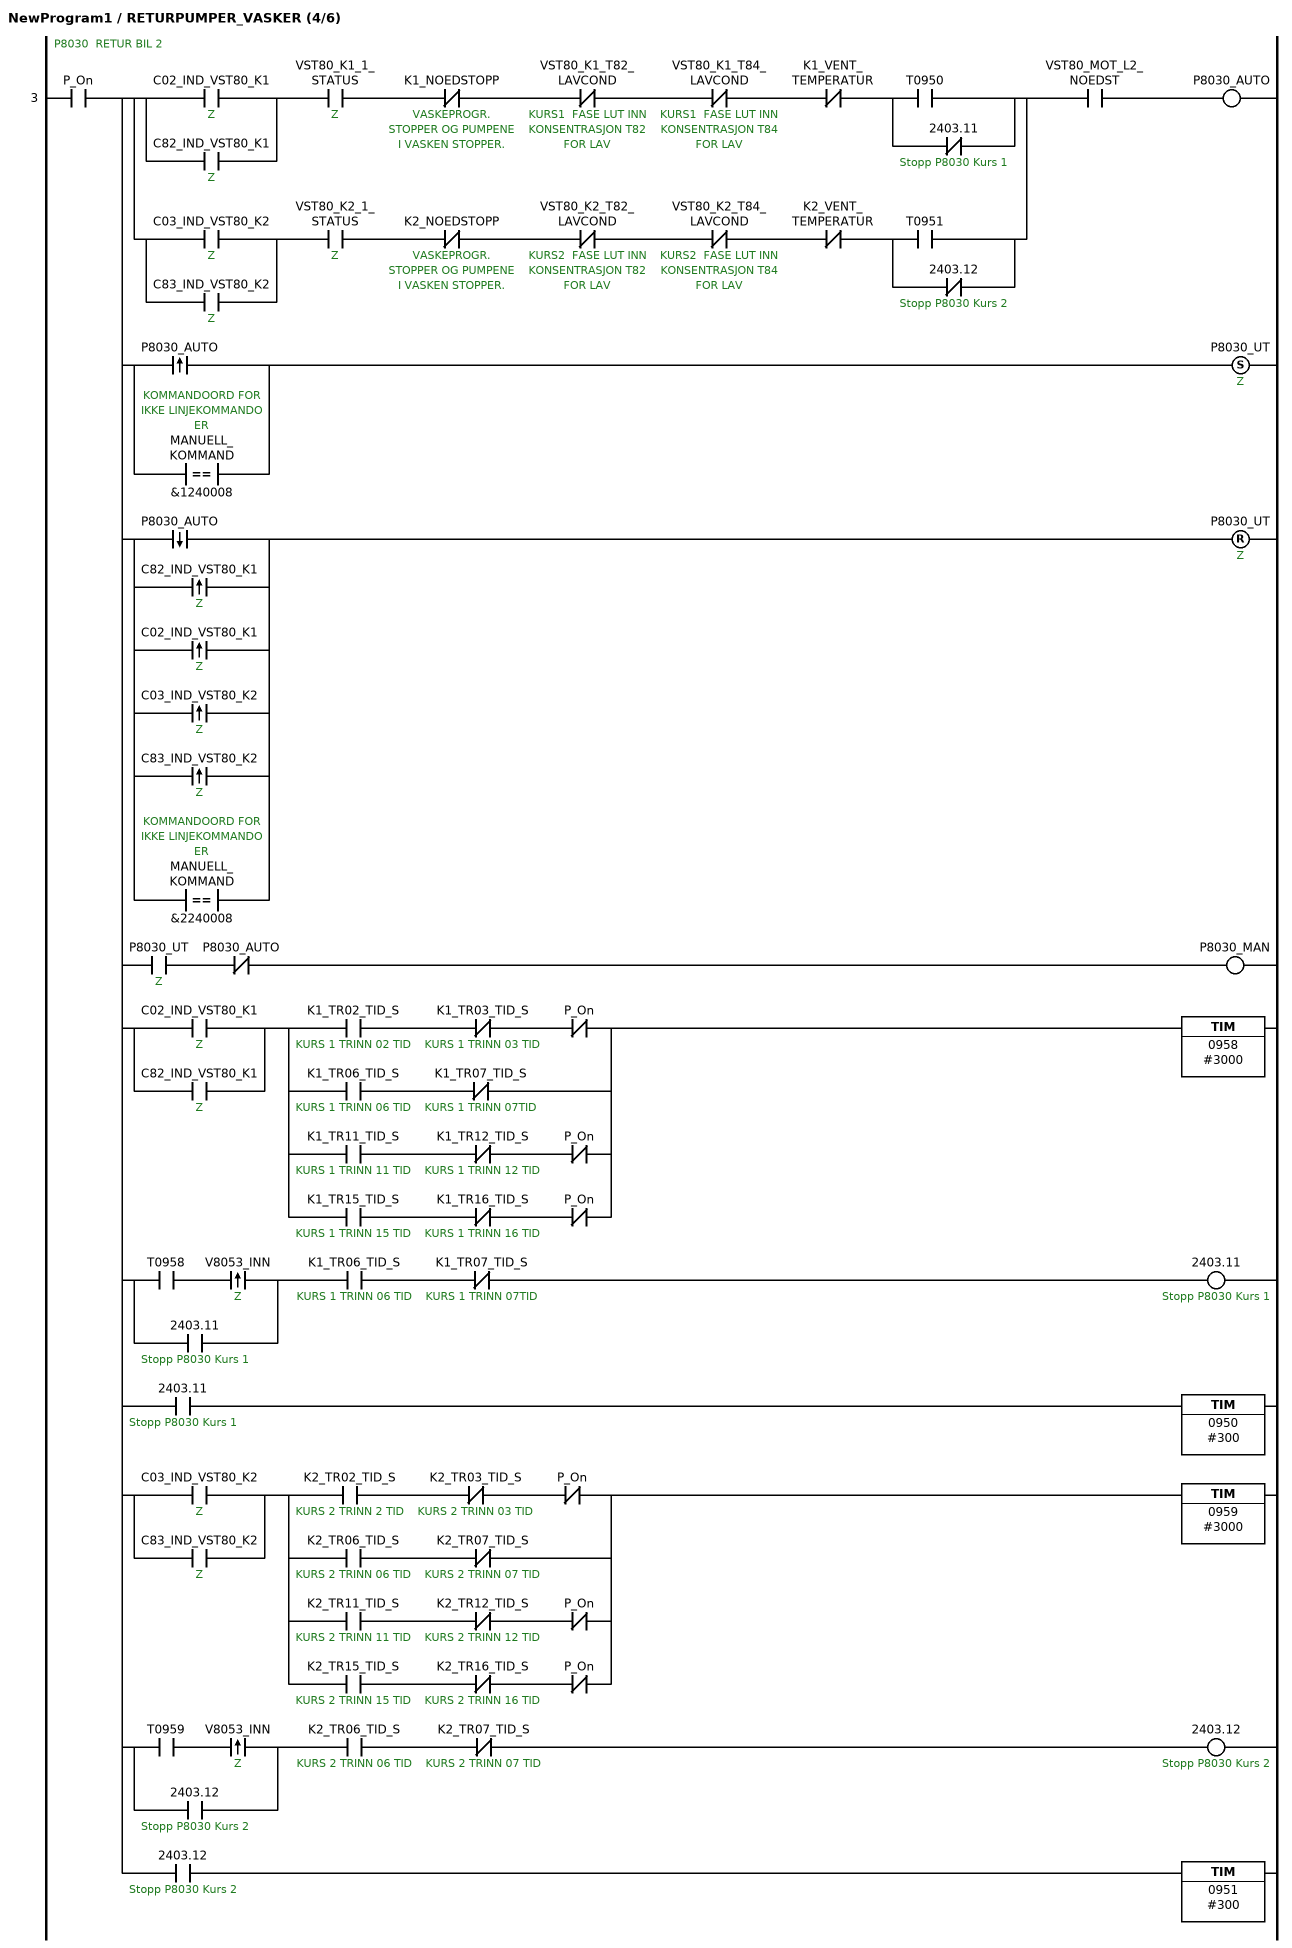
; rung 3: P8030  RETUR BIL 2
LD P_On
OUT TR0
LD C02_IND_VST80_K1  ; Z
OR C82_IND_VST80_K1  ; Z
AND VST80_K1_1_STATUS  ; Z
ANDNOT K1_NOEDSTOPP  ; VASKEPROGR. STOPPER OG PUMPENE I VASKEN STOPPER.
ANDNOT VST80_K1_T82_LAVCOND  ; KURS1  FASE LUT INN KONSENTRASJON T82 FOR LAV
ANDNOT VST80_K1_T84_LAVCOND  ; KURS1  FASE LUT INN KONSENTRASJON T84 FOR LAV
ANDNOT K1_VENT_TEMPERATUR
LD T0950
ORNOT 2403.11  ; Stopp P8030 Kurs 1
ANDLD
LD C03_IND_VST80_K2  ; Z
OR C83_IND_VST80_K2  ; Z
AND VST80_K2_1_STATUS  ; Z
ANDNOT K2_NOEDSTOPP  ; VASKEPROGR. STOPPER OG PUMPENE I VASKEN STOPPER.
ANDNOT VST80_K2_T82_LAVCOND  ; KURS2  FASE LUT INN KONSENTRASJON T82 FOR LAV
ANDNOT VST80_K2_T84_LAVCOND  ; KURS2  FASE LUT INN KONSENTRASJON T84 FOR LAV
ANDNOT K2_VENT_TEMPERATUR
LD T0951
ORNOT 2403.12  ; Stopp P8030 Kurs 2
ANDLD
ORLD
ANDLD
AND VST80_MOT_L2_NOEDST
OUT P8030_AUTO
LD TR0
@LD P8030_AUTO
OR=L(301) MANUELL_KOMMAND &1240008  ; KOMMANDOORD FOR IKKE LINJEKOMMANDOER
ANDLD
SET P8030_UT  ; Z
LD TR0
%LD P8030_AUTO
@OR C82_IND_VST80_K1  ; Z
@OR C02_IND_VST80_K1  ; Z
@OR C03_IND_VST80_K2  ; Z
@OR C83_IND_VST80_K2  ; Z
OR=L(301) MANUELL_KOMMAND &2240008  ; KOMMANDOORD FOR IKKE LINJEKOMMANDOER
ANDLD
RSET P8030_UT  ; Z
LD TR0
AND P8030_UT  ; Z
ANDNOT P8030_AUTO
OUT P8030_MAN
LD TR0
LD C02_IND_VST80_K1  ; Z
OR C82_IND_VST80_K1  ; Z
ANDLD
LD K1_TR02_TID_S  ; KURS 1 TRINN 02 TID
ANDNOT K1_TR03_TID_S  ; KURS 1 TRINN 03 TID
ANDNOT P_On
LD K1_TR06_TID_S  ; KURS 1 TRINN 06 TID
ANDNOT K1_TR07_TID_S  ; KURS 1 TRINN 07TID
ORLD
LD K1_TR11_TID_S  ; KURS 1 TRINN 11 TID
ANDNOT K1_TR12_TID_S  ; KURS 1 TRINN 12 TID
ANDNOT P_On
ORLD
LD K1_TR15_TID_S  ; KURS 1 TRINN 15 TID
ANDNOT K1_TR16_TID_S  ; KURS 1 TRINN 16 TID
ANDNOT P_On
ORLD
ANDLD
TIM 0958 #3000
LD TR0
LD T0958
@AND V8053_INN  ; Z
OR 2403.11  ; Stopp P8030 Kurs 1
ANDLD
AND K1_TR06_TID_S  ; KURS 1 TRINN 06 TID
ANDNOT K1_TR07_TID_S  ; KURS 1 TRINN 07TID
OUT 2403.11  ; Stopp P8030 Kurs 1
LD TR0
AND 2403.11  ; Stopp P8030 Kurs 1
TIM 0950 #300
LD TR0
LD C03_IND_VST80_K2  ; Z
OR C83_IND_VST80_K2  ; Z
ANDLD
LD K2_TR02_TID_S  ; KURS 2 TRINN 2 TID
ANDNOT K2_TR03_TID_S  ; KURS 2 TRINN 03 TID
ANDNOT P_On
LD K2_TR06_TID_S  ; KURS 2 TRINN 06 TID
ANDNOT K2_TR07_TID_S  ; KURS 2 TRINN 07 TID
ORLD
LD K2_TR11_TID_S  ; KURS 2 TRINN 11 TID
ANDNOT K2_TR12_TID_S  ; KURS 2 TRINN 12 TID
ANDNOT P_On
ORLD
LD K2_TR15_TID_S  ; KURS 2 TRINN 15 TID
ANDNOT K2_TR16_TID_S  ; KURS 2 TRINN 16 TID
ANDNOT P_On
ORLD
ANDLD
TIM 0959 #3000
LD TR0
LD T0959
@AND V8053_INN  ; Z
OR 2403.12  ; Stopp P8030 Kurs 2
ANDLD
AND K2_TR06_TID_S  ; KURS 2 TRINN 06 TID
ANDNOT K2_TR07_TID_S  ; KURS 2 TRINN 07 TID
OUT 2403.12  ; Stopp P8030 Kurs 2
LD TR0
AND 2403.12  ; Stopp P8030 Kurs 2
TIM 0951 #300

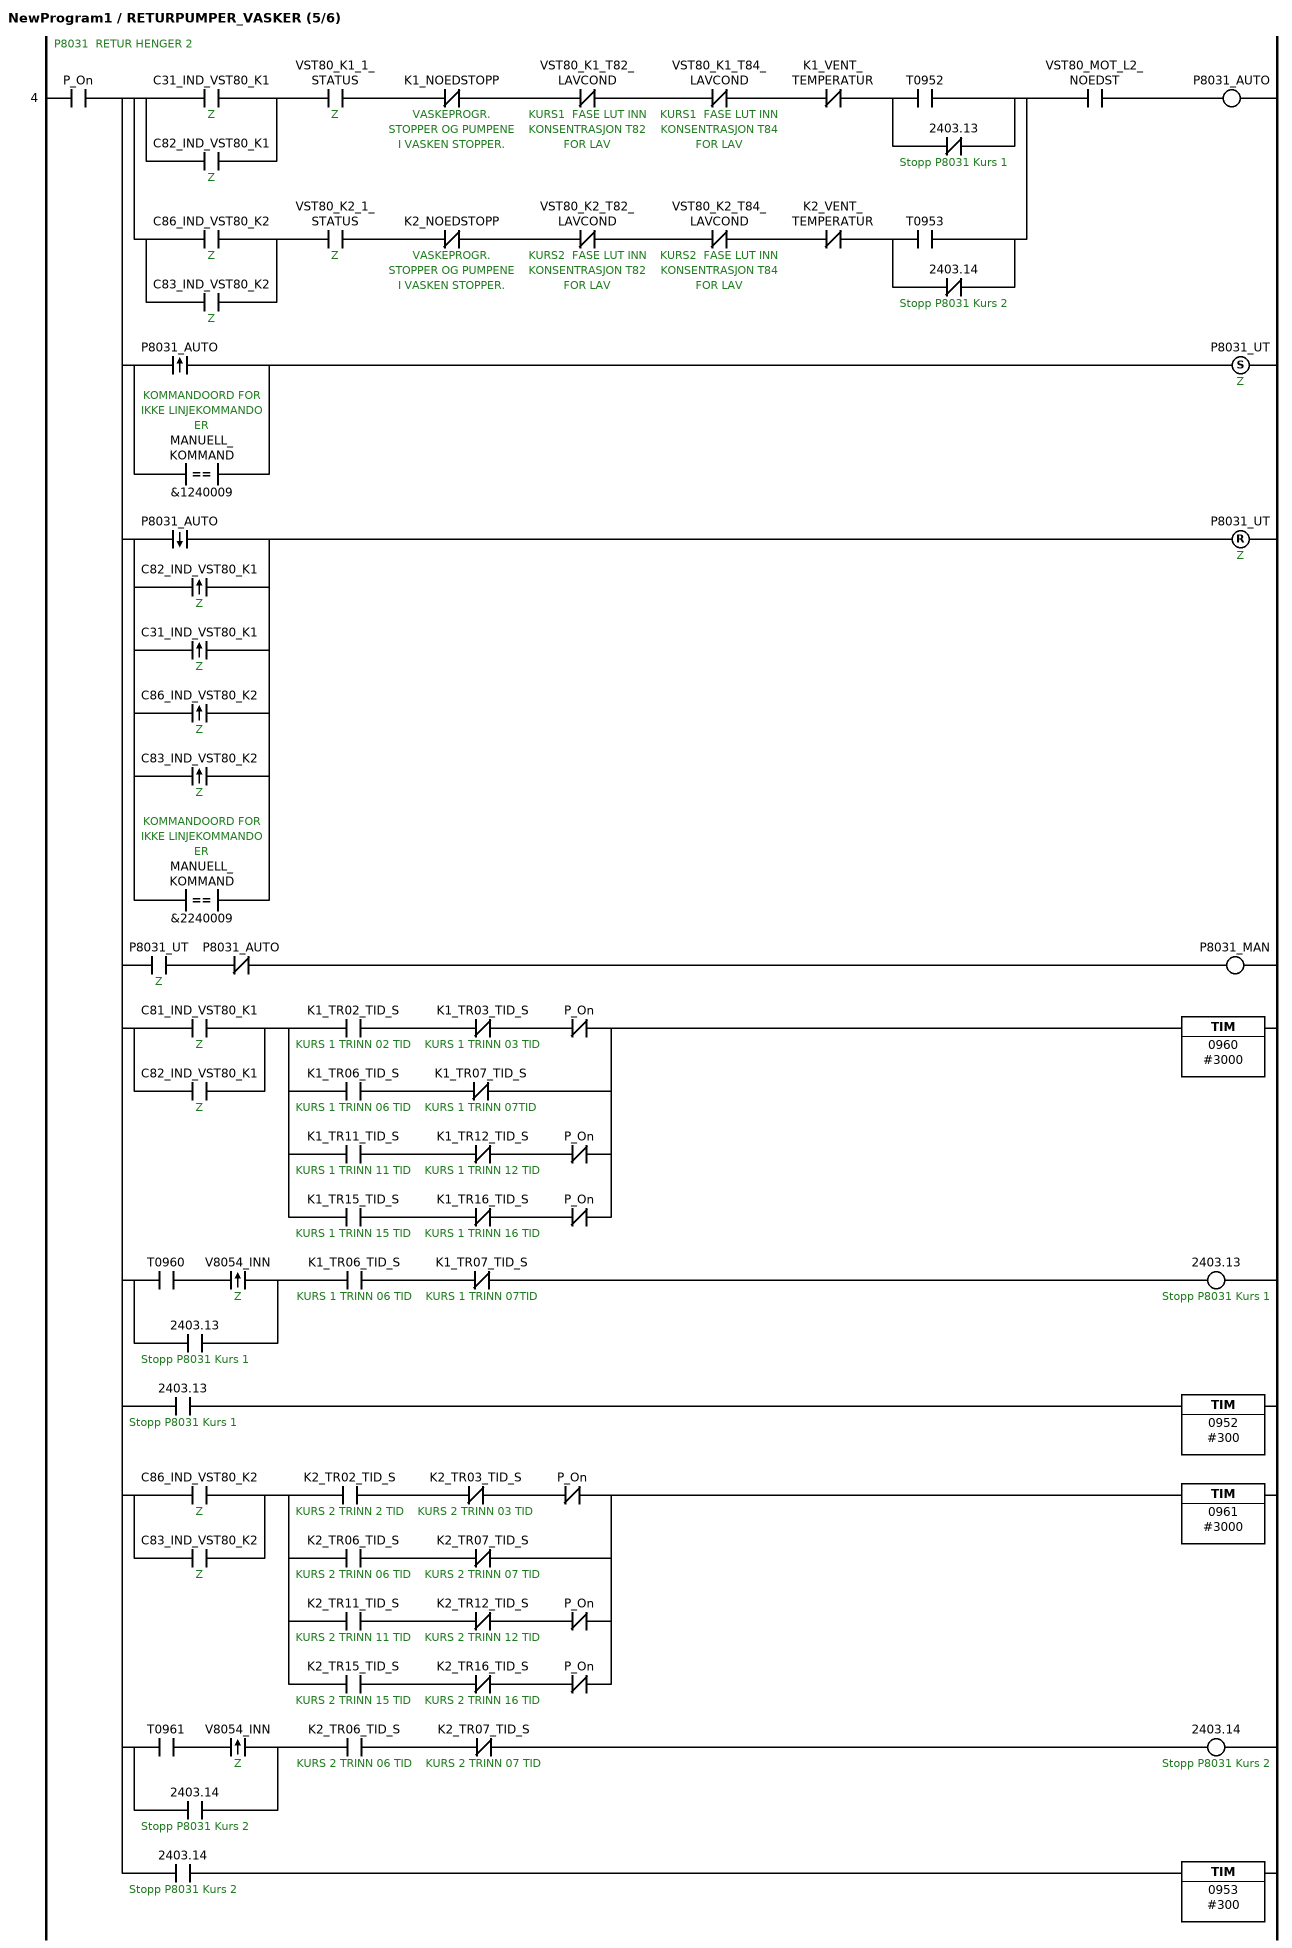
; rung 4: P8031  RETUR HENGER 2
LD P_On
OUT TR0
LD C31_IND_VST80_K1  ; Z
OR C82_IND_VST80_K1  ; Z
AND VST80_K1_1_STATUS  ; Z
ANDNOT K1_NOEDSTOPP  ; VASKEPROGR. STOPPER OG PUMPENE I VASKEN STOPPER.
ANDNOT VST80_K1_T82_LAVCOND  ; KURS1  FASE LUT INN KONSENTRASJON T82 FOR LAV
ANDNOT VST80_K1_T84_LAVCOND  ; KURS1  FASE LUT INN KONSENTRASJON T84 FOR LAV
ANDNOT K1_VENT_TEMPERATUR
LD T0952
ORNOT 2403.13  ; Stopp P8031 Kurs 1
ANDLD
LD C86_IND_VST80_K2  ; Z
OR C83_IND_VST80_K2  ; Z
AND VST80_K2_1_STATUS  ; Z
ANDNOT K2_NOEDSTOPP  ; VASKEPROGR. STOPPER OG PUMPENE I VASKEN STOPPER.
ANDNOT VST80_K2_T82_LAVCOND  ; KURS2  FASE LUT INN KONSENTRASJON T82 FOR LAV
ANDNOT VST80_K2_T84_LAVCOND  ; KURS2  FASE LUT INN KONSENTRASJON T84 FOR LAV
ANDNOT K2_VENT_TEMPERATUR
LD T0953
ORNOT 2403.14  ; Stopp P8031 Kurs 2
ANDLD
ORLD
ANDLD
AND VST80_MOT_L2_NOEDST
OUT P8031_AUTO
LD TR0
@LD P8031_AUTO
OR=L(301) MANUELL_KOMMAND &1240009  ; KOMMANDOORD FOR IKKE LINJEKOMMANDOER
ANDLD
SET P8031_UT  ; Z
LD TR0
%LD P8031_AUTO
@OR C82_IND_VST80_K1  ; Z
@OR C31_IND_VST80_K1  ; Z
@OR C86_IND_VST80_K2  ; Z
@OR C83_IND_VST80_K2  ; Z
OR=L(301) MANUELL_KOMMAND &2240009  ; KOMMANDOORD FOR IKKE LINJEKOMMANDOER
ANDLD
RSET P8031_UT  ; Z
LD TR0
AND P8031_UT  ; Z
ANDNOT P8031_AUTO
OUT P8031_MAN
LD TR0
LD C81_IND_VST80_K1  ; Z
OR C82_IND_VST80_K1  ; Z
ANDLD
LD K1_TR02_TID_S  ; KURS 1 TRINN 02 TID
ANDNOT K1_TR03_TID_S  ; KURS 1 TRINN 03 TID
ANDNOT P_On
LD K1_TR06_TID_S  ; KURS 1 TRINN 06 TID
ANDNOT K1_TR07_TID_S  ; KURS 1 TRINN 07TID
ORLD
LD K1_TR11_TID_S  ; KURS 1 TRINN 11 TID
ANDNOT K1_TR12_TID_S  ; KURS 1 TRINN 12 TID
ANDNOT P_On
ORLD
LD K1_TR15_TID_S  ; KURS 1 TRINN 15 TID
ANDNOT K1_TR16_TID_S  ; KURS 1 TRINN 16 TID
ANDNOT P_On
ORLD
ANDLD
TIM 0960 #3000
LD TR0
LD T0960
@AND V8054_INN  ; Z
OR 2403.13  ; Stopp P8031 Kurs 1
ANDLD
AND K1_TR06_TID_S  ; KURS 1 TRINN 06 TID
ANDNOT K1_TR07_TID_S  ; KURS 1 TRINN 07TID
OUT 2403.13  ; Stopp P8031 Kurs 1
LD TR0
AND 2403.13  ; Stopp P8031 Kurs 1
TIM 0952 #300
LD TR0
LD C86_IND_VST80_K2  ; Z
OR C83_IND_VST80_K2  ; Z
ANDLD
LD K2_TR02_TID_S  ; KURS 2 TRINN 2 TID
ANDNOT K2_TR03_TID_S  ; KURS 2 TRINN 03 TID
ANDNOT P_On
LD K2_TR06_TID_S  ; KURS 2 TRINN 06 TID
ANDNOT K2_TR07_TID_S  ; KURS 2 TRINN 07 TID
ORLD
LD K2_TR11_TID_S  ; KURS 2 TRINN 11 TID
ANDNOT K2_TR12_TID_S  ; KURS 2 TRINN 12 TID
ANDNOT P_On
ORLD
LD K2_TR15_TID_S  ; KURS 2 TRINN 15 TID
ANDNOT K2_TR16_TID_S  ; KURS 2 TRINN 16 TID
ANDNOT P_On
ORLD
ANDLD
TIM 0961 #3000
LD TR0
LD T0961
@AND V8054_INN  ; Z
OR 2403.14  ; Stopp P8031 Kurs 2
ANDLD
AND K2_TR06_TID_S  ; KURS 2 TRINN 06 TID
ANDNOT K2_TR07_TID_S  ; KURS 2 TRINN 07 TID
OUT 2403.14  ; Stopp P8031 Kurs 2
LD TR0
AND 2403.14  ; Stopp P8031 Kurs 2
TIM 0953 #300

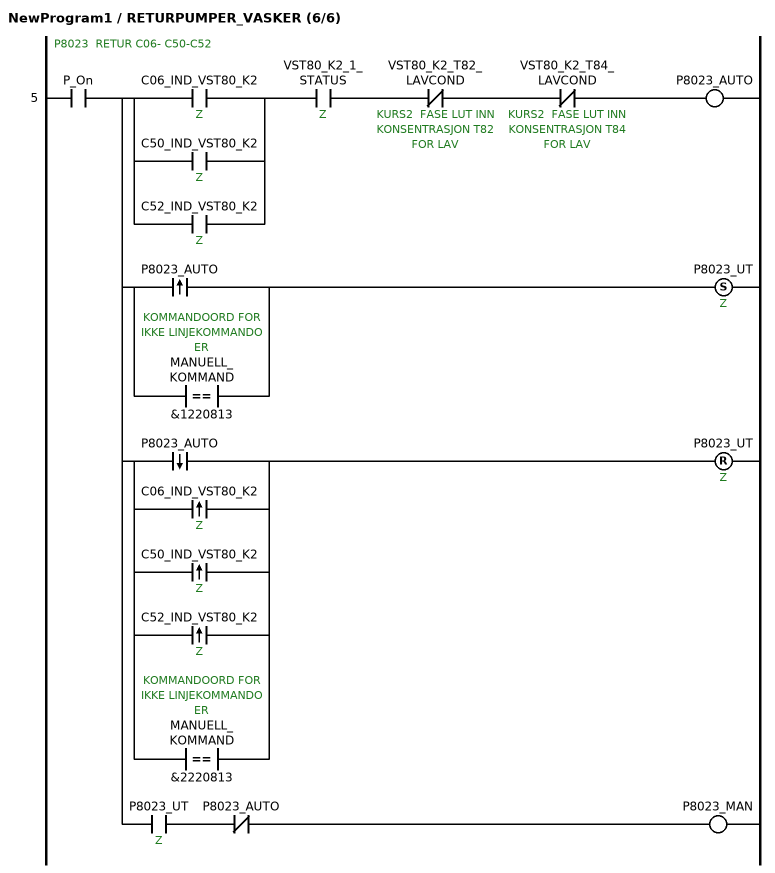
; rung 5: P8023  RETUR C06- C50-C52
LD P_On
OUT TR0
LD C06_IND_VST80_K2  ; Z
OR C50_IND_VST80_K2  ; Z
OR C52_IND_VST80_K2  ; Z
ANDLD
AND VST80_K2_1_STATUS  ; Z
ANDNOT VST80_K2_T82_LAVCOND  ; KURS2  FASE LUT INN KONSENTRASJON T82 FOR LAV
ANDNOT VST80_K2_T84_LAVCOND  ; KURS2  FASE LUT INN KONSENTRASJON T84 FOR LAV
OUT P8023_AUTO
LD TR0
@LD P8023_AUTO
OR=L(301) MANUELL_KOMMAND &1220813  ; KOMMANDOORD FOR IKKE LINJEKOMMANDOER
ANDLD
SET P8023_UT  ; Z
LD TR0
%LD P8023_AUTO
@OR C06_IND_VST80_K2  ; Z
@OR C50_IND_VST80_K2  ; Z
@OR C52_IND_VST80_K2  ; Z
OR=L(301) MANUELL_KOMMAND &2220813  ; KOMMANDOORD FOR IKKE LINJEKOMMANDOER
ANDLD
RSET P8023_UT  ; Z
LD TR0
AND P8023_UT  ; Z
ANDNOT P8023_AUTO
OUT P8023_MAN

### Section VENTILER_VASKFORDELING

